Yaskawa INFORM job: A_ROOF_UPPER_0614_2_PAINT_52.JBI

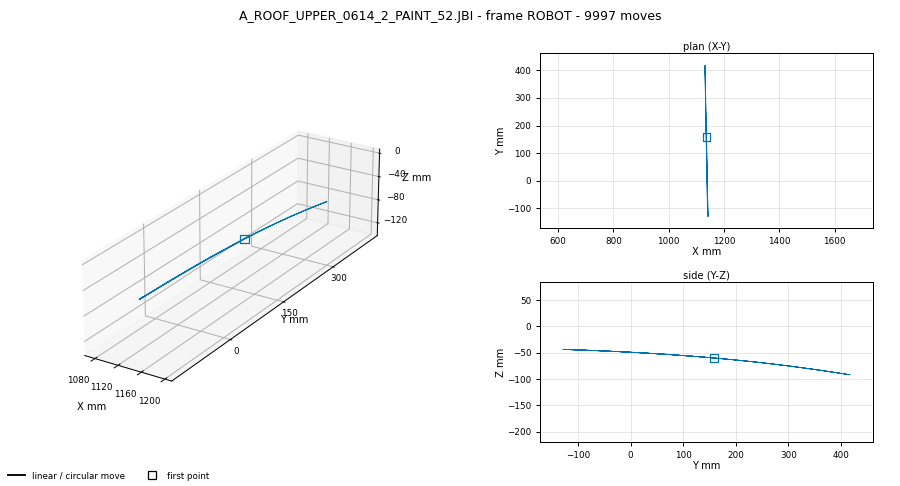
[picture p0: tool path of A_ROOF_UPPER_0614_2_PAINT_52.JBI in frame ROBOT, 9997 of 9997 moves have a stored position in this frame; points joined in program order, loops and branches not executed]
/JOB
//NAME A_ROOF_UPPER_0614_2_PAINT52
//POS
///NPOS 9997,0,0,0,0,0
///TOOL 1
///USER 0
///POSTYPE ROBOT
///RECTAN
///RCONF 1,0,0,0,0,0,0,0,0,0,0,0,0,0,0,0,0,0,0,0,0,0,0,0
C00000=1136.806,158.945,-59.840,-178.647,7.166,148.946
C00001=1136.811,158.695,-59.818,-178.650,7.165,148.946
C00002=1136.815,158.447,-59.796,-178.653,7.163,148.946
C00003=1136.820,158.198,-59.775,-178.656,7.160,148.947
C00004=1136.825,157.948,-59.753,-178.658,7.158,148.947
C00005=1136.829,157.680,-59.730,-178.662,7.156,148.947
C00006=1136.835,157.410,-59.707,-178.665,7.153,148.948
C00007=1136.840,157.141,-59.683,-178.668,7.152,148.948
C00008=1136.845,156.872,-59.660,-178.671,7.149,148.948
C00009=1136.850,156.623,-59.639,-178.674,7.147,148.949
C00010=1136.855,156.374,-59.617,-178.677,7.144,148.949
C00011=1136.859,156.125,-59.595,-178.679,7.143,148.949
C00012=1136.864,155.876,-59.573,-178.682,7.141,148.950
C00013=1136.869,155.627,-59.552,-178.685,7.139,148.950
C00014=1136.873,155.379,-59.531,-178.688,7.136,148.950
C00015=1136.878,155.129,-59.510,-178.690,7.135,148.951
C00016=1136.883,154.880,-59.488,-178.694,7.132,148.951
C00017=1136.887,154.632,-59.467,-178.696,7.131,148.951
C00018=1136.892,154.382,-59.445,-178.699,7.129,148.952
C00019=1136.897,154.133,-59.424,-178.702,7.126,148.952
C00020=1136.901,153.884,-59.403,-178.705,7.124,148.952
C00021=1136.906,153.635,-59.381,-178.707,7.123,148.953
C00022=1136.911,153.386,-59.359,-178.711,7.120,148.953
C00023=1136.916,153.137,-59.338,-178.713,7.118,148.953
C00024=1136.921,152.888,-59.317,-178.716,7.115,148.954
C00025=1136.925,152.639,-59.296,-178.719,7.114,148.954
C00026=1136.929,152.390,-59.274,-178.722,7.112,148.954
C00027=1136.934,152.141,-59.253,-178.725,7.110,148.955
C00028=1136.939,151.892,-59.232,-178.728,7.108,148.955
C00029=1136.944,151.643,-59.211,-178.730,7.106,148.955
C00030=1136.948,151.393,-59.190,-178.732,7.104,148.956
C00031=1136.953,151.144,-59.168,-178.736,7.102,148.956
C00032=1136.958,150.895,-59.147,-178.739,7.100,148.956
C00033=1136.962,150.647,-59.126,-178.741,7.098,148.957
C00034=1136.968,150.398,-59.105,-178.744,7.095,148.957
C00035=1136.972,150.148,-59.083,-178.747,7.094,148.957
C00036=1136.977,149.899,-59.062,-178.749,7.092,148.958
C00037=1136.982,149.650,-59.042,-178.753,7.089,148.958
C00038=1136.986,149.401,-59.020,-178.755,7.088,148.958
C00039=1136.992,149.152,-58.999,-178.758,7.086,148.959
C00040=1136.996,148.903,-58.979,-178.761,7.083,148.959
C00041=1137.000,148.654,-58.957,-178.764,7.081,148.959
C00042=1137.005,148.405,-58.936,-178.766,7.080,148.960
C00043=1137.010,148.156,-58.915,-178.770,7.077,148.960
C00044=1137.015,147.907,-58.894,-178.772,7.075,148.960
C00045=1137.020,147.658,-58.873,-178.775,7.073,148.961
C00046=1137.024,147.409,-58.852,-178.777,7.072,148.961
C00047=1137.029,147.159,-58.831,-178.781,7.069,148.961
C00048=1137.033,146.911,-58.810,-178.783,7.067,148.962
C00049=1137.038,146.661,-58.789,-178.786,7.066,148.962
C00050=1137.043,146.412,-58.768,-178.790,7.063,148.963
C00051=1137.048,146.163,-58.748,-178.792,7.062,148.963
C00052=1137.053,145.914,-58.727,-178.794,7.059,148.963
C00053=1137.057,145.665,-58.706,-178.797,7.058,148.963
C00054=1137.062,145.416,-58.685,-178.800,7.055,148.964
C00055=1137.067,145.167,-58.664,-178.803,7.054,148.964
C00056=1137.071,144.917,-58.643,-178.806,7.052,148.965
C00057=1137.076,144.668,-58.623,-178.809,7.049,148.965
C00058=1137.081,144.419,-58.602,-178.812,7.048,148.965
C00059=1137.085,144.170,-58.581,-178.814,7.046,148.966
C00060=1137.090,143.922,-58.560,-178.817,7.044,148.966
C00061=1137.095,143.673,-58.539,-178.820,7.041,148.966
C00062=1137.100,143.423,-58.518,-178.823,7.040,148.967
C00063=1137.104,143.174,-58.498,-178.826,7.038,148.967
C00064=1137.110,142.925,-58.477,-178.828,7.036,148.967
C00065=1137.114,142.676,-58.457,-178.832,7.034,148.968
C00066=1137.119,142.427,-58.436,-178.834,7.032,148.968
C00067=1137.124,142.178,-58.415,-178.837,7.030,148.968
C00068=1137.129,141.929,-58.394,-178.839,7.028,148.969
C00069=1137.133,141.680,-58.374,-178.843,7.026,148.969
C00070=1137.138,141.431,-58.354,-178.845,7.024,148.970
C00071=1137.143,141.182,-58.333,-178.848,7.022,148.970
C00072=1137.147,140.933,-58.312,-178.851,7.021,148.970
C00073=1137.152,140.683,-58.291,-178.854,7.018,148.971
C00074=1137.157,140.434,-58.271,-178.857,7.016,148.971
C00075=1137.161,140.185,-58.250,-178.859,7.014,148.971
C00076=1137.166,139.936,-58.230,-178.862,7.013,148.972
C00077=1137.171,139.687,-58.210,-178.865,7.010,148.972
C00078=1137.176,139.438,-58.189,-178.868,7.009,148.972
C00079=1137.181,139.188,-58.169,-178.871,7.007,148.973
C00080=1137.185,138.939,-58.148,-178.873,7.005,148.973
C00081=1137.190,138.690,-58.128,-178.877,7.003,148.974
C00082=1137.195,138.441,-58.107,-178.879,7.001,148.974
C00083=1137.199,138.192,-58.086,-178.882,6.999,148.974
C00084=1137.204,137.943,-58.067,-178.885,6.998,148.975
C00085=1137.209,137.693,-58.046,-178.887,6.995,148.975
C00086=1137.214,137.444,-58.025,-178.890,6.993,148.975
C00087=1137.218,137.196,-58.005,-178.893,6.991,148.976
C00088=1137.223,136.946,-57.984,-178.896,6.990,148.976
C00089=1137.228,136.697,-57.964,-178.898,6.988,148.977
C00090=1137.232,136.448,-57.944,-178.901,6.986,148.977
C00091=1137.237,136.199,-57.924,-178.905,6.984,148.977
C00092=1137.243,135.950,-57.903,-178.907,6.982,148.978
C00093=1137.247,135.701,-57.883,-178.910,6.980,148.978
C00094=1137.252,135.452,-57.863,-178.913,6.979,148.978
C00095=1137.256,135.203,-57.843,-178.915,6.977,148.979
C00096=1137.261,134.953,-57.823,-178.919,6.974,148.979
C00097=1137.266,134.704,-57.802,-178.921,6.972,148.979
C00098=1137.271,134.455,-57.782,-178.924,6.971,148.980
C00099=1137.275,134.205,-57.762,-178.926,6.969,148.980
C00100=1137.280,133.957,-57.742,-178.929,6.967,148.981
C00101=1137.285,133.708,-57.722,-178.932,6.965,148.981
C00102=1137.290,133.458,-57.701,-178.935,6.963,148.981
C00103=1137.295,133.209,-57.681,-178.938,6.961,148.982
C00104=1137.300,132.960,-57.661,-178.941,6.960,148.982
C00105=1137.304,132.711,-57.641,-178.943,6.958,148.983
C00106=1137.309,132.461,-57.621,-178.947,6.955,148.983
C00107=1137.314,132.213,-57.601,-178.949,6.954,148.983
C00108=1137.319,131.964,-57.580,-178.952,6.952,148.984
C00109=1137.324,131.695,-57.559,-178.955,6.950,148.984
C00110=1137.329,131.427,-57.538,-178.958,6.948,148.985
C00111=1137.334,131.158,-57.516,-178.961,6.946,148.985
C00112=1137.339,130.890,-57.495,-178.964,6.944,148.985
C00113=1137.344,130.640,-57.475,-178.967,6.942,148.986
C00114=1137.348,130.391,-57.455,-178.970,6.940,148.986
C00115=1137.354,130.142,-57.435,-178.972,6.939,148.986
C00116=1137.359,129.893,-57.414,-178.975,6.937,148.987
C00117=1137.363,129.643,-57.395,-178.978,6.935,148.987
C00118=1137.368,129.394,-57.374,-178.980,6.933,148.988
C00119=1137.373,129.145,-57.355,-178.984,6.931,148.988
C00120=1137.378,128.896,-57.335,-178.987,6.929,148.988
C00121=1137.382,128.647,-57.315,-178.989,6.928,148.989
C00122=1137.387,128.397,-57.295,-178.992,6.926,148.989
C00123=1137.392,128.148,-57.276,-178.995,6.924,148.990
C00124=1137.397,127.900,-57.256,-178.997,6.923,148.990
C00125=1137.402,127.650,-57.236,-179.000,6.921,148.990
C00126=1137.406,127.401,-57.216,-179.003,6.918,148.991
C00127=1137.411,127.152,-57.196,-179.006,6.917,148.991
C00128=1137.416,126.903,-57.177,-179.009,6.915,148.992
C00129=1137.421,126.653,-57.157,-179.012,6.913,148.992
C00130=1137.425,126.404,-57.137,-179.014,6.912,148.992
C00131=1137.431,126.155,-57.117,-179.017,6.910,148.993
C00132=1137.435,125.906,-57.098,-179.020,6.908,148.993
C00133=1137.439,125.657,-57.078,-179.023,6.907,148.994
C00134=1137.444,125.408,-57.059,-179.026,6.904,148.994
C00135=1137.449,125.159,-57.039,-179.029,6.902,148.994
C00136=1137.454,124.909,-57.019,-179.031,6.901,148.995
C00137=1137.459,124.659,-57.000,-179.034,6.899,148.995
C00138=1137.464,124.411,-56.980,-179.037,6.897,148.996
C00139=1137.468,124.162,-56.960,-179.039,6.896,148.996
C00140=1137.473,123.912,-56.940,-179.042,6.894,148.996
C00141=1137.478,123.664,-56.922,-179.045,6.892,148.997
C00142=1137.483,123.414,-56.902,-179.048,6.890,148.997
C00143=1137.488,123.165,-56.883,-179.051,6.888,148.998
C00144=1137.492,122.916,-56.862,-179.054,6.886,148.998
C00145=1137.497,122.667,-56.843,-179.056,6.885,148.998
C00146=1137.502,122.418,-56.824,-179.059,6.883,148.999
C00147=1137.506,122.168,-56.804,-179.062,6.881,148.999
C00148=1137.511,121.919,-56.785,-179.065,6.880,149.000
C00149=1137.517,121.670,-56.766,-179.067,6.878,149.000
C00150=1137.521,121.420,-56.746,-179.070,6.876,149.000
C00151=1137.526,121.171,-56.726,-179.073,6.875,149.001
C00152=1137.531,120.922,-56.708,-179.076,6.873,149.001
C00153=1137.535,120.673,-56.688,-179.079,6.870,149.002
C00154=1137.541,120.424,-56.669,-179.082,6.869,149.002
C00155=1137.545,120.174,-56.649,-179.084,6.867,149.002
C00156=1137.550,119.926,-56.630,-179.087,6.865,149.003
C00157=1137.555,119.676,-56.611,-179.090,6.864,149.003
C00158=1137.560,119.427,-56.591,-179.092,6.862,149.004
C00159=1137.565,119.178,-56.572,-179.095,6.860,149.004
C00160=1137.569,118.929,-56.553,-179.098,6.859,149.004
C00161=1137.574,118.680,-56.533,-179.101,6.857,149.005
C00162=1137.579,118.430,-56.514,-179.103,6.855,149.005
C00163=1137.584,118.182,-56.495,-179.106,6.853,149.006
C00164=1137.588,117.932,-56.475,-179.109,6.852,149.006
C00165=1137.594,117.683,-56.456,-179.112,6.850,149.006
C00166=1137.598,117.433,-56.438,-179.114,6.848,149.007
C00167=1137.603,117.184,-56.418,-179.117,6.847,149.007
C00168=1137.608,116.935,-56.399,-179.120,6.844,149.008
C00169=1137.612,116.686,-56.380,-179.123,6.843,149.008
C00170=1137.617,116.437,-56.360,-179.126,6.841,149.008
C00171=1137.622,116.187,-56.341,-179.129,6.839,149.009
C00172=1137.627,115.938,-56.323,-179.131,6.838,149.009
C00173=1137.632,115.688,-56.303,-179.134,6.836,149.010
C00174=1137.637,115.439,-56.284,-179.137,6.834,149.010
C00175=1137.641,115.190,-56.265,-179.139,6.832,149.011
C00176=1137.647,114.941,-56.245,-179.143,6.831,149.011
C00177=1137.651,114.691,-56.227,-179.145,6.829,149.012
C00178=1137.656,114.443,-56.208,-179.148,6.828,149.012
C00179=1137.662,114.194,-56.188,-179.151,6.826,149.012
C00180=1137.666,113.944,-56.170,-179.154,6.824,149.013
C00181=1137.671,113.695,-56.151,-179.156,6.823,149.013
C00182=1137.675,113.446,-56.132,-179.159,6.821,149.014
C00183=1137.681,113.197,-56.112,-179.162,6.819,149.014
C00184=1137.685,112.947,-56.094,-179.165,6.818,149.014
C00185=1137.690,112.698,-56.075,-179.167,6.816,149.015
C00186=1137.694,112.449,-56.056,-179.170,6.814,149.015
C00187=1137.700,112.199,-56.037,-179.173,6.813,149.016
C00188=1137.704,111.951,-56.018,-179.175,6.811,149.016
C00189=1137.710,111.701,-56.000,-179.178,6.809,149.016
C00190=1137.714,111.452,-55.981,-179.181,6.808,149.017
C00191=1137.719,111.203,-55.961,-179.184,6.806,149.017
C00192=1137.724,110.953,-55.943,-179.187,6.805,149.018
C00193=1137.729,110.704,-55.924,-179.190,6.803,149.018
C00194=1137.733,110.455,-55.906,-179.192,6.801,149.019
C00195=1137.739,110.206,-55.886,-179.195,6.800,149.019
C00196=1137.743,109.956,-55.868,-179.198,6.798,149.020
C00197=1137.748,109.707,-55.849,-179.200,6.796,149.020
C00198=1137.753,109.458,-55.830,-179.203,6.795,149.020
C00199=1137.758,109.208,-55.811,-179.206,6.793,149.021
C00200=1137.763,108.960,-55.792,-179.209,6.791,149.021
C00201=1137.768,108.711,-55.774,-179.211,6.789,149.022
C00202=1137.772,108.461,-55.755,-179.214,6.788,149.022
C00203=1137.777,108.212,-55.737,-179.217,6.786,149.022
C00204=1137.782,107.962,-55.718,-179.220,6.785,149.023
C00205=1137.787,107.713,-55.699,-179.223,6.783,149.023
C00206=1137.792,107.464,-55.681,-179.226,6.781,149.024
C00207=1137.797,107.214,-55.661,-179.228,6.780,149.024
C00208=1137.801,106.965,-55.643,-179.231,6.778,149.025
C00209=1137.806,106.717,-55.625,-179.234,6.776,149.025
C00210=1137.812,106.467,-55.606,-179.236,6.775,149.026
C00211=1137.816,106.217,-55.588,-179.239,6.773,149.026
C00212=1137.821,105.969,-55.569,-179.242,6.771,149.026
C00213=1137.826,105.700,-55.549,-179.245,6.770,149.027
C00214=1137.831,105.431,-55.529,-179.248,6.768,149.027
C00215=1137.837,105.163,-55.509,-179.251,6.766,149.028
C00216=1137.842,104.895,-55.489,-179.254,6.764,149.028
C00217=1137.846,104.646,-55.471,-179.257,6.763,149.029
C00218=1137.852,104.396,-55.453,-179.260,6.761,149.029
C00219=1137.856,104.147,-55.434,-179.263,6.760,149.030
C00220=1137.861,103.898,-55.416,-179.265,6.758,149.030
C00221=1137.867,103.648,-55.397,-179.268,6.757,149.030
C00222=1137.871,103.398,-55.379,-179.270,6.755,149.031
C00223=1137.876,103.150,-55.360,-179.273,6.754,149.031
C00224=1137.880,102.901,-55.342,-179.276,6.752,149.032
C00225=1137.885,102.652,-55.324,-179.278,6.750,149.032
C00226=1137.891,102.402,-55.305,-179.282,6.749,149.033
C00227=1137.895,102.152,-55.287,-179.284,6.747,149.033
C00228=1137.900,101.904,-55.268,-179.287,6.746,149.034
C00229=1137.905,101.654,-55.250,-179.290,6.744,149.034
C00230=1137.910,101.405,-55.232,-179.293,6.742,149.034
C00231=1137.915,101.155,-55.214,-179.295,6.741,149.035
C00232=1137.920,100.906,-55.196,-179.298,6.739,149.035
C00233=1137.925,100.657,-55.178,-179.301,6.737,149.036
C00234=1137.929,100.408,-55.159,-179.304,6.736,149.036
C00235=1137.934,100.159,-55.141,-179.307,6.734,149.037
C00236=1137.939,99.909,-55.123,-179.309,6.733,149.037
C00237=1137.944,99.660,-55.104,-179.312,6.732,149.038
C00238=1137.949,99.410,-55.086,-179.314,6.730,149.038
C00239=1137.954,99.161,-55.068,-179.317,6.728,149.038
C00240=1137.959,98.912,-55.050,-179.320,6.727,149.039
C00241=1137.964,98.663,-55.032,-179.323,6.725,149.039
C00242=1137.968,98.413,-55.014,-179.326,6.724,149.040
C00243=1137.973,98.164,-54.996,-179.329,6.722,149.040
C00244=1137.978,97.915,-54.978,-179.331,6.720,149.041
C00245=1137.983,97.666,-54.960,-179.334,6.719,149.041
C00246=1137.988,97.416,-54.942,-179.337,6.717,149.042
C00247=1137.993,97.167,-54.923,-179.339,6.716,149.042
C00248=1137.998,96.918,-54.905,-179.342,6.715,149.043
C00249=1138.003,96.668,-54.887,-179.345,6.713,149.043
C00250=1138.008,96.419,-54.869,-179.348,6.712,149.043
C00251=1138.012,96.169,-54.851,-179.350,6.710,149.044
C00252=1138.017,95.920,-54.833,-179.353,6.708,149.044
C00253=1138.022,95.671,-54.815,-179.356,6.707,149.045
C00254=1138.027,95.422,-54.797,-179.359,6.705,149.045
C00255=1138.032,95.173,-54.779,-179.362,6.704,149.046
C00256=1138.037,94.924,-54.761,-179.364,6.703,149.046
C00257=1138.042,94.674,-54.744,-179.367,6.701,149.047
C00258=1138.047,94.425,-54.726,-179.369,6.699,149.047
C00259=1138.051,94.175,-54.707,-179.372,6.698,149.047
C00260=1138.056,93.926,-54.689,-179.375,6.696,149.048
C00261=1138.061,93.676,-54.672,-179.378,6.695,149.048
C00262=1138.066,93.427,-54.654,-179.381,6.693,149.049
C00263=1138.071,93.177,-54.636,-179.384,6.691,149.049
C00264=1138.076,92.929,-54.619,-179.386,6.691,149.050
C00265=1138.080,92.679,-54.601,-179.388,6.689,149.050
C00266=1138.085,92.430,-54.583,-179.391,6.687,149.051
C00267=1138.090,92.181,-54.565,-179.394,6.686,149.051
C00268=1138.096,91.931,-54.548,-179.397,6.684,149.052
C00269=1138.100,91.682,-54.530,-179.400,6.683,149.052
C00270=1138.105,91.433,-54.512,-179.403,6.681,149.053
C00271=1138.110,91.184,-54.494,-179.405,6.680,149.053
C00272=1138.115,90.934,-54.476,-179.408,6.678,149.053
C00273=1138.120,90.685,-54.458,-179.411,6.677,149.054
C00274=1138.125,90.436,-54.441,-179.413,6.675,149.054
C00275=1138.130,90.186,-54.424,-179.416,6.674,149.055
C00276=1138.135,89.937,-54.406,-179.419,6.672,149.055
C00277=1138.140,89.688,-54.388,-179.422,6.670,149.056
C00278=1138.145,89.438,-54.371,-179.424,6.670,149.056
C00279=1138.150,89.189,-54.353,-179.427,6.668,149.057
C00280=1138.154,88.940,-54.335,-179.430,6.667,149.057
C00281=1138.159,88.690,-54.318,-179.433,6.665,149.058
C00282=1138.164,88.441,-54.300,-179.435,6.663,149.058
C00283=1138.169,88.191,-54.283,-179.438,6.662,149.058
C00284=1138.174,87.942,-54.265,-179.441,6.661,149.059
C00285=1138.178,87.693,-54.247,-179.443,6.659,149.060
C00286=1138.184,87.443,-54.230,-179.446,6.658,149.060
C00287=1138.188,87.194,-54.212,-179.449,6.656,149.060
C00288=1138.194,86.944,-54.195,-179.452,6.654,149.061
C00289=1138.199,86.695,-54.177,-179.455,6.653,149.061
C00290=1138.203,86.446,-54.160,-179.457,6.652,149.062
C00291=1138.208,86.196,-54.142,-179.460,6.651,149.062
C00292=1138.214,85.947,-54.125,-179.462,6.649,149.063
C00293=1138.218,85.699,-54.108,-179.465,6.647,149.063
C00294=1138.223,85.449,-54.091,-179.468,6.646,149.064
C00295=1138.228,85.200,-54.073,-179.471,6.645,149.064
C00296=1138.233,84.950,-54.055,-179.473,6.644,149.065
C00297=1138.238,84.701,-54.038,-179.476,6.642,149.065
C00298=1138.243,84.451,-54.021,-179.479,6.640,149.065
C00299=1138.248,84.202,-54.003,-179.482,6.639,149.066
C00300=1138.252,83.952,-53.986,-179.484,6.638,149.067
C00301=1138.257,83.703,-53.969,-179.487,6.636,149.067
C00302=1138.263,83.454,-53.951,-179.490,6.635,149.067
C00303=1138.267,83.205,-53.935,-179.492,6.633,149.068
C00304=1138.272,82.956,-53.917,-179.496,6.632,149.068
C00305=1138.277,82.706,-53.899,-179.498,6.631,149.069
C00306=1138.282,82.456,-53.883,-179.501,6.629,149.069
C00307=1138.287,82.207,-53.865,-179.503,6.628,149.070
C00308=1138.291,81.958,-53.848,-179.506,6.626,149.070
C00309=1138.297,81.708,-53.831,-179.509,6.625,149.071
C00310=1138.302,81.459,-53.813,-179.511,6.624,149.071
C00311=1138.307,81.210,-53.796,-179.514,6.622,149.072
C00312=1138.312,80.960,-53.779,-179.517,6.620,149.072
C00313=1138.316,80.711,-53.762,-179.520,6.619,149.073
C00314=1138.322,80.462,-53.745,-179.522,6.618,149.073
C00315=1138.327,80.212,-53.728,-179.525,6.617,149.074
C00316=1138.331,79.963,-53.711,-179.528,6.615,149.074
C00317=1138.337,79.694,-53.692,-179.531,6.614,149.075
C00318=1138.342,79.427,-53.674,-179.534,6.612,149.075
C00319=1138.347,79.158,-53.655,-179.537,6.611,149.076
C00320=1138.353,78.889,-53.636,-179.540,6.609,149.076
C00321=1138.358,78.640,-53.620,-179.542,6.607,149.077
C00322=1138.363,78.390,-53.603,-179.545,6.607,149.077
C00323=1138.367,78.141,-53.586,-179.548,6.605,149.078
C00324=1138.373,77.891,-53.569,-179.551,6.604,149.078
C00325=1138.377,77.643,-53.552,-179.553,6.602,149.079
C00326=1138.383,77.393,-53.535,-179.555,6.601,149.079
C00327=1138.387,77.144,-53.518,-179.559,6.600,149.080
C00328=1138.392,76.894,-53.501,-179.561,6.598,149.080
C00329=1138.397,76.645,-53.484,-179.564,6.597,149.081
C00330=1138.403,76.395,-53.467,-179.566,6.596,149.081
C00331=1138.407,76.146,-53.451,-179.569,6.594,149.081
C00332=1138.412,75.896,-53.434,-179.572,6.593,149.082
C00333=1138.417,75.648,-53.416,-179.575,6.591,149.082
C00334=1138.422,75.398,-53.400,-179.577,6.590,149.083
C00335=1138.427,75.149,-53.382,-179.580,6.589,149.083
C00336=1138.432,74.900,-53.366,-179.583,6.587,149.084
C00337=1138.436,74.650,-53.349,-179.585,6.586,149.084
C00338=1138.442,74.400,-53.332,-179.588,6.585,149.085
C00339=1138.446,74.151,-53.315,-179.591,6.583,149.085
C00340=1138.452,73.902,-53.299,-179.594,6.582,149.086
C00341=1138.456,73.652,-53.282,-179.596,6.581,149.086
C00342=1138.461,73.403,-53.265,-179.599,6.579,149.087
C00343=1138.467,73.154,-53.248,-179.602,6.578,149.087
C00344=1138.471,72.904,-53.232,-179.605,6.576,149.088
C00345=1138.476,72.655,-53.215,-179.607,6.576,149.088
C00346=1138.481,72.406,-53.198,-179.610,6.574,149.089
C00347=1138.486,72.156,-53.182,-179.613,6.572,149.089
C00348=1138.491,71.906,-53.165,-179.615,6.572,149.090
C00349=1138.496,71.657,-53.149,-179.618,6.570,149.090
C00350=1138.501,71.408,-53.132,-179.621,6.568,149.091
C00351=1138.505,71.158,-53.115,-179.623,6.568,149.091
C00352=1138.511,70.909,-53.098,-179.626,6.566,149.092
C00353=1138.516,70.660,-53.082,-179.629,6.565,149.092
C00354=1138.521,70.411,-53.065,-179.632,6.563,149.093
C00355=1138.526,70.161,-53.048,-179.634,6.562,149.093
C00356=1138.531,69.911,-53.032,-179.637,6.561,149.094
C00357=1138.536,69.662,-53.016,-179.640,6.559,149.094
C00358=1138.540,69.413,-52.999,-179.642,6.558,149.095
C00359=1138.546,69.164,-52.982,-179.645,6.557,149.095
C00360=1138.551,68.914,-52.966,-179.648,6.555,149.096
C00361=1138.555,68.664,-52.950,-179.650,6.555,149.096
C00362=1138.561,68.415,-52.933,-179.653,6.553,149.097
C00363=1138.566,68.165,-52.916,-179.656,6.552,149.097
C00364=1138.571,67.917,-52.900,-179.658,6.551,149.098
C00365=1138.575,67.667,-52.883,-179.661,6.549,149.098
C00366=1138.580,67.417,-52.867,-179.664,6.547,149.099
C00367=1138.585,67.168,-52.851,-179.666,6.547,149.099
C00368=1138.590,66.918,-52.834,-179.669,6.545,149.100
C00369=1138.596,66.669,-52.818,-179.672,6.544,149.100
C00370=1138.600,66.420,-52.801,-179.674,6.543,149.101
C00371=1138.605,66.171,-52.785,-179.677,6.542,149.101
C00372=1138.610,65.921,-52.768,-179.680,6.540,149.102
C00373=1138.615,65.671,-52.752,-179.682,6.539,149.102
C00374=1138.620,65.422,-52.735,-179.685,6.538,149.103
C00375=1138.625,65.172,-52.719,-179.688,6.536,149.103
C00376=1138.630,64.923,-52.703,-179.690,6.535,149.104
C00377=1138.635,64.674,-52.687,-179.693,6.534,149.104
C00378=1138.640,64.424,-52.671,-179.696,6.532,149.105
C00379=1138.645,64.175,-52.654,-179.698,6.532,149.105
C00380=1138.650,63.926,-52.638,-179.701,6.530,149.106
C00381=1138.655,63.676,-52.622,-179.704,6.529,149.106
C00382=1138.660,63.427,-52.606,-179.706,6.528,149.107
C00383=1138.665,63.177,-52.589,-179.709,6.526,149.107
C00384=1138.670,62.928,-52.573,-179.712,6.524,149.108
C00385=1138.675,62.678,-52.557,-179.715,6.524,149.108
C00386=1138.680,62.429,-52.541,-179.717,6.522,149.109
C00387=1138.685,62.180,-52.524,-179.720,6.521,149.109
C00388=1138.690,61.930,-52.508,-179.723,6.520,149.110
C00389=1138.694,61.681,-52.492,-179.725,6.519,149.110
C00390=1138.700,61.431,-52.476,-179.728,6.518,149.111
C00391=1138.704,61.182,-52.459,-179.730,6.516,149.111
C00392=1138.710,60.932,-52.444,-179.734,6.515,149.112
C00393=1138.715,60.683,-52.428,-179.736,6.514,149.112
C00394=1138.720,60.433,-52.412,-179.739,6.512,149.113
C00395=1138.725,60.184,-52.396,-179.742,6.511,149.113
C00396=1138.729,59.935,-52.379,-179.744,6.510,149.114
C00397=1138.735,59.685,-52.364,-179.747,6.509,149.114
C00398=1138.739,59.436,-52.347,-179.749,6.508,149.115
C00399=1138.745,59.186,-52.331,-179.752,6.506,149.115
C00400=1138.750,58.937,-52.316,-179.755,6.505,149.116
C00401=1138.755,58.687,-52.299,-179.757,6.504,149.116
C00402=1138.760,58.438,-52.284,-179.760,6.503,149.117
C00403=1138.764,58.189,-52.267,-179.763,6.501,149.117
C00404=1138.770,57.939,-52.251,-179.765,6.500,149.118
C00405=1138.775,57.690,-52.236,-179.768,6.499,149.118
C00406=1138.780,57.440,-52.219,-179.770,6.498,149.119
C00407=1138.785,57.191,-52.204,-179.773,6.496,149.119
C00408=1138.789,56.941,-52.188,-179.776,6.495,149.120
C00409=1138.794,56.692,-52.172,-179.779,6.494,149.120
C00410=1138.800,56.443,-52.156,-179.781,6.493,149.121
C00411=1138.804,56.193,-52.140,-179.784,6.492,149.121
C00412=1138.810,55.943,-52.125,-179.787,6.491,149.122
C00413=1138.815,55.695,-52.108,-179.789,6.490,149.122
C00414=1138.820,55.444,-52.092,-179.792,6.488,149.123
C00415=1138.825,55.195,-52.077,-179.795,6.487,149.123
C00416=1138.830,54.946,-52.061,-179.797,6.486,149.124
C00417=1138.834,54.696,-52.045,-179.800,6.484,149.124
C00418=1138.839,54.447,-52.030,-179.802,6.484,149.125
C00419=1138.845,54.198,-52.014,-179.805,6.482,149.125
C00420=1138.850,53.948,-51.998,-179.808,6.481,149.126
C00421=1138.855,53.679,-51.981,-179.811,6.480,149.127
C00422=1138.861,53.411,-51.964,-179.813,6.479,149.127
C00423=1138.866,53.142,-51.947,-179.817,6.477,149.128
C00424=1138.871,52.874,-51.931,-179.819,6.476,149.128
C00425=1138.876,52.624,-51.915,-179.822,6.475,149.129
C00426=1138.881,52.374,-51.899,-179.825,6.474,149.129
C00427=1138.887,52.125,-51.883,-179.827,6.473,149.130
C00428=1138.891,51.875,-51.868,-179.830,6.471,149.130
C00429=1138.896,51.626,-51.852,-179.832,6.471,149.131
C00430=1138.901,51.377,-51.836,-179.835,6.469,149.131
C00431=1138.907,51.128,-51.821,-179.838,6.467,149.132
C00432=1138.911,50.878,-51.805,-179.840,6.467,149.132
C00433=1138.916,50.628,-51.790,-179.843,6.465,149.133
C00434=1138.921,50.379,-51.774,-179.845,6.464,149.133
C00435=1138.927,50.130,-51.759,-179.849,6.463,149.134
C00436=1138.932,49.880,-51.743,-179.851,6.462,149.134
C00437=1138.936,49.630,-51.728,-179.854,6.461,149.135
C00438=1138.942,49.381,-51.712,-179.856,6.460,149.135
C00439=1138.947,49.132,-51.696,-179.859,6.459,149.136
C00440=1138.951,48.882,-51.681,-179.861,6.458,149.136
C00441=1138.956,48.632,-51.665,-179.864,6.456,149.137
C00442=1138.962,48.383,-51.650,-179.867,6.455,149.137
C00443=1138.966,48.134,-51.635,-179.869,6.454,149.138
C00444=1138.971,47.884,-51.619,-179.873,6.453,149.139
C00445=1138.977,47.634,-51.603,-179.875,6.452,149.139
C00446=1138.981,47.385,-51.588,-179.877,6.450,149.139
C00447=1138.987,47.136,-51.573,-179.880,6.449,149.140
C00448=1138.992,46.887,-51.557,-179.883,6.448,149.141
C00449=1138.996,46.637,-51.542,-179.885,6.447,149.141
C00450=1139.002,46.387,-51.526,-179.888,6.446,149.141
C00451=1139.006,46.138,-51.511,-179.890,6.445,149.142
C00452=1139.012,45.888,-51.496,-179.893,6.444,149.143
C00453=1139.017,45.639,-51.481,-179.895,6.443,149.143
C00454=1139.021,45.389,-51.465,-179.899,6.441,149.144
C00455=1139.027,45.140,-51.450,-179.901,6.441,149.144
C00456=1139.031,44.891,-51.435,-179.903,6.439,149.145
C00457=1139.037,44.641,-51.419,-179.906,6.439,149.145
C00458=1139.042,44.392,-51.404,-179.909,6.437,149.146
C00459=1139.047,44.142,-51.389,-179.911,6.436,149.146
C00460=1139.052,43.893,-51.374,-179.914,6.435,149.147
C00461=1139.056,43.643,-51.358,-179.916,6.434,149.147
C00462=1139.062,43.393,-51.343,-179.919,6.432,149.148
C00463=1139.067,43.144,-51.328,-179.922,6.432,149.148
C00464=1139.072,42.894,-51.313,-179.925,6.430,149.149
C00465=1139.077,42.645,-51.298,-179.927,6.429,149.149
C00466=1139.082,42.396,-51.282,-179.930,6.428,149.150
C00467=1139.087,42.147,-51.267,-179.932,6.427,149.150
C00468=1139.093,41.897,-51.253,-179.935,6.426,149.151
C00469=1139.097,41.647,-51.237,-179.938,6.425,149.151
C00470=1139.102,41.398,-51.222,-179.940,6.424,149.152
C00471=1139.107,41.148,-51.207,-179.943,6.423,149.153
C00472=1139.112,40.898,-51.192,-179.946,6.422,149.153
C00473=1139.117,40.649,-51.177,-179.948,6.421,149.153
C00474=1139.122,40.400,-51.161,-179.951,6.419,149.154
C00475=1139.127,40.150,-51.147,-179.953,6.419,149.155
C00476=1139.133,39.901,-51.131,-179.956,6.417,149.155
C00477=1139.138,39.651,-51.117,-179.959,6.417,149.156
C00478=1139.143,39.402,-51.101,-179.961,6.415,149.156
C00479=1139.148,39.153,-51.086,-179.964,6.414,149.157
C00480=1139.153,38.903,-51.072,-179.967,6.413,149.157
C00481=1139.158,38.654,-51.057,-179.969,6.412,149.158
C00482=1139.163,38.404,-51.042,-179.972,6.410,149.158
C00483=1139.168,38.154,-51.026,-179.974,6.410,149.159
C00484=1139.172,37.905,-51.011,-179.977,6.409,149.159
C00485=1139.178,37.655,-50.996,-179.979,6.407,149.160
C00486=1139.183,37.406,-50.981,-179.982,6.407,149.160
C00487=1139.188,37.156,-50.967,-179.985,6.405,149.161
C00488=1139.193,36.906,-50.952,-179.987,6.405,149.161
C00489=1139.198,36.657,-50.937,-179.990,6.403,149.162
C00490=1139.203,36.408,-50.922,-179.992,6.402,149.162
C00491=1139.208,36.158,-50.907,-179.995,6.401,149.163
C00492=1139.213,35.908,-50.892,-179.998,6.400,149.164
C00493=1139.218,35.659,-50.877,179.999,6.399,149.164
C00494=1139.223,35.409,-50.863,179.997,6.398,149.165
C00495=1139.228,35.160,-50.848,179.995,6.397,149.165
C00496=1139.234,34.910,-50.833,179.992,6.396,149.166
C00497=1139.239,34.661,-50.818,179.989,6.395,149.166
C00498=1139.243,34.411,-50.803,179.986,6.394,149.167
C00499=1139.248,34.162,-50.789,179.984,6.393,149.167
C00500=1139.254,33.912,-50.774,179.981,6.392,149.168
C00501=1139.259,33.663,-50.760,179.979,6.391,149.168
C00502=1139.264,33.414,-50.745,179.977,6.390,149.169
C00503=1139.270,33.164,-50.730,179.973,6.389,149.169
C00504=1139.275,32.915,-50.716,179.971,6.388,149.170
C00505=1139.279,32.665,-50.701,179.969,6.386,149.170
C00506=1139.284,32.416,-50.686,179.966,6.386,149.171
C00507=1139.290,32.166,-50.671,179.963,6.384,149.172
C00508=1139.295,31.917,-50.656,179.961,6.383,149.172
C00509=1139.299,31.667,-50.642,179.958,6.383,149.173
C00510=1139.304,31.418,-50.627,179.956,6.381,149.173
C00511=1139.310,31.168,-50.612,179.953,6.381,149.174
C00512=1139.315,30.918,-50.598,179.950,6.379,149.174
C00513=1139.319,30.669,-50.583,179.948,6.378,149.175
C00514=1139.324,30.419,-50.569,179.945,6.377,149.175
C00515=1139.329,30.170,-50.554,179.943,6.376,149.176
C00516=1139.336,29.920,-50.540,179.940,6.376,149.176
C00517=1139.340,29.671,-50.525,179.937,6.374,149.177
C00518=1139.345,29.421,-50.511,179.935,6.373,149.177
C00519=1139.350,29.172,-50.496,179.932,6.372,149.178
C00520=1139.355,28.922,-50.482,179.930,6.371,149.179
C00521=1139.360,28.673,-50.467,179.927,6.371,149.179
C00522=1139.365,28.423,-50.452,179.924,6.369,149.180
C00523=1139.370,28.173,-50.438,179.922,6.368,149.180
C00524=1139.376,27.924,-50.424,179.919,6.367,149.181
C00525=1139.381,27.655,-50.408,179.917,6.366,149.181
C00526=1139.386,27.387,-50.393,179.914,6.365,149.182
C00527=1139.392,27.117,-50.377,179.911,6.364,149.182
C00528=1139.398,26.848,-50.361,179.908,6.363,149.183
C00529=1139.403,26.598,-50.347,179.906,6.362,149.184
C00530=1139.407,26.349,-50.333,179.903,6.361,149.184
C00531=1139.413,26.100,-50.319,179.900,6.360,149.185
C00532=1139.418,25.851,-50.304,179.898,6.359,149.185
C00533=1139.423,25.601,-50.290,179.895,6.358,149.186
C00534=1139.428,25.351,-50.275,179.893,6.357,149.186
C00535=1139.433,25.101,-50.261,179.891,6.357,149.187
C00536=1139.437,24.852,-50.247,179.888,6.355,149.187
C00537=1139.444,24.602,-50.232,179.885,6.354,149.188
C00538=1139.449,24.353,-50.218,179.882,6.353,149.188
C00539=1139.454,24.103,-50.204,179.880,6.352,149.189
C00540=1139.459,23.853,-50.189,179.878,6.352,149.189
C00541=1139.464,23.604,-50.175,179.875,6.350,149.190
C00542=1139.469,23.355,-50.161,179.872,6.350,149.191
C00543=1139.474,23.105,-50.147,179.870,6.349,149.191
C00544=1139.479,22.855,-50.133,179.867,6.347,149.191
C00545=1139.484,22.605,-50.118,179.865,6.347,149.192
C00546=1139.490,22.356,-50.105,179.862,6.346,149.193
C00547=1139.495,22.107,-50.090,179.860,6.344,149.193
C00548=1139.499,21.857,-50.076,179.857,6.344,149.194
C00549=1139.504,21.607,-50.062,179.855,6.343,149.194
C00550=1139.509,21.358,-50.047,179.852,6.342,149.195
C00551=1139.515,21.109,-50.034,179.849,6.341,149.195
C00552=1139.519,20.859,-50.020,179.847,6.339,149.196
C00553=1139.524,20.609,-50.006,179.844,6.339,149.196
C00554=1139.530,20.360,-49.992,179.842,6.338,149.197
C00555=1139.535,20.111,-49.977,179.839,6.336,149.197
C00556=1139.540,19.861,-49.963,179.836,6.336,149.198
C00557=1139.545,19.611,-49.949,179.834,6.335,149.199
C00558=1139.550,19.362,-49.935,179.831,6.334,149.199
C00559=1139.555,19.113,-49.921,179.829,6.333,149.200
C00560=1139.560,18.862,-49.907,179.827,6.332,149.200
C00561=1139.566,18.613,-49.893,179.823,6.331,149.201
C00562=1139.571,18.364,-49.879,179.821,6.330,149.201
C00563=1139.576,18.114,-49.865,179.819,6.329,149.202
C00564=1139.581,17.864,-49.850,179.816,6.328,149.202
C00565=1139.586,17.615,-49.837,179.814,6.327,149.203
C00566=1139.591,17.366,-49.823,179.811,6.327,149.204
C00567=1139.596,17.115,-49.809,179.809,6.326,149.204
C00568=1139.601,16.866,-49.795,179.806,6.324,149.204
C00569=1139.606,16.617,-49.781,179.803,6.324,149.205
C00570=1139.611,16.367,-49.767,179.801,6.323,149.206
C00571=1139.616,16.118,-49.753,179.798,6.322,149.206
C00572=1139.621,15.868,-49.740,179.796,6.321,149.207
C00573=1139.626,15.618,-49.726,179.794,6.320,149.207
C00574=1139.632,15.369,-49.712,179.790,6.319,149.208
C00575=1139.637,15.119,-49.697,179.788,6.318,149.208
C00576=1139.642,14.869,-49.684,179.786,6.317,149.209
C00577=1139.647,14.620,-49.670,179.783,6.316,149.209
C00578=1139.652,14.371,-49.656,179.781,6.315,149.210
C00579=1139.658,14.121,-49.643,179.778,6.315,149.211
C00580=1139.663,13.871,-49.629,179.776,6.314,149.211
C00581=1139.667,13.622,-49.615,179.773,6.313,149.212
C00582=1139.673,13.372,-49.602,179.770,6.312,149.212
C00583=1139.678,13.123,-49.588,179.768,6.311,149.213
C00584=1139.683,12.873,-49.573,179.765,6.310,149.213
C00585=1139.688,12.623,-49.560,179.763,6.309,149.214
C00586=1139.693,12.374,-49.546,179.761,6.308,149.214
C00587=1139.698,12.125,-49.532,179.758,6.308,149.215
C00588=1139.704,11.875,-49.519,179.755,6.306,149.215
C00589=1139.708,11.625,-49.505,179.753,6.306,149.216
C00590=1139.713,11.376,-49.491,179.750,6.305,149.217
C00591=1139.719,11.126,-49.478,179.748,6.304,149.217
C00592=1139.724,10.877,-49.464,179.745,6.303,149.218
C00593=1139.729,10.627,-49.451,179.743,6.302,149.218
C00594=1139.734,10.378,-49.437,179.741,6.301,149.219
C00595=1139.739,10.128,-49.423,179.737,6.300,149.219
C00596=1139.744,9.879,-49.410,179.735,6.299,149.220
C00597=1139.749,9.629,-49.396,179.733,6.299,149.220
C00598=1139.754,9.379,-49.382,179.730,6.298,149.221
C00599=1139.759,9.130,-49.369,179.728,6.297,149.221
C00600=1139.765,8.880,-49.355,179.725,6.296,149.222
C00601=1139.770,8.631,-49.341,179.723,6.295,149.223
C00602=1139.775,8.381,-49.329,179.720,6.294,149.223
C00603=1139.780,8.132,-49.315,179.717,6.293,149.224
C00604=1139.785,7.881,-49.301,179.715,6.292,149.224
C00605=1139.790,7.633,-49.288,179.713,6.292,149.225
C00606=1139.796,7.382,-49.274,179.710,6.290,149.225
C00607=1139.800,7.134,-49.261,179.708,6.290,149.226
C00608=1139.806,6.883,-49.247,179.705,6.289,149.226
C00609=1139.811,6.634,-49.234,179.703,6.288,149.227
C00610=1139.816,6.384,-49.220,179.700,6.287,149.227
C00611=1139.822,6.135,-49.207,179.697,6.286,149.228
C00612=1139.826,5.885,-49.194,179.695,6.286,149.229
C00613=1139.832,5.636,-49.180,179.693,6.285,149.229
C00614=1139.837,5.386,-49.166,179.690,6.284,149.230
C00615=1139.842,5.137,-49.153,179.687,6.283,149.230
C00616=1139.847,4.886,-49.140,179.685,6.282,149.231
C00617=1139.852,4.638,-49.127,179.683,6.281,149.231
C00618=1139.857,4.387,-49.113,179.680,6.281,149.232
C00619=1139.862,4.138,-49.100,179.677,6.279,149.232
C00620=1139.867,3.888,-49.086,179.675,6.279,149.233
C00621=1139.872,3.639,-49.074,179.672,6.278,149.234
C00622=1139.878,3.389,-49.060,179.670,6.277,149.234
C00623=1139.882,3.140,-49.047,179.667,6.276,149.235
C00624=1139.888,2.890,-49.033,179.665,6.275,149.235
C00625=1139.893,2.640,-49.020,179.663,6.275,149.236
C00626=1139.898,2.391,-49.007,179.660,6.274,149.236
C00627=1139.903,2.141,-48.994,179.658,6.273,149.237
C00628=1139.909,1.892,-48.980,179.655,6.272,149.237
C00629=1139.913,1.622,-48.966,179.652,6.271,149.238
C00630=1139.919,1.352,-48.952,179.650,6.270,149.238
C00631=1139.925,1.083,-48.938,179.647,6.269,149.239
C00632=1139.930,0.814,-48.923,179.644,6.269,149.240
C00633=1139.936,0.564,-48.910,179.642,6.268,149.240
C00634=1139.941,0.314,-48.897,179.639,6.266,149.241
C00635=1139.946,0.065,-48.884,179.637,6.266,149.241
C00636=1139.951,-0.185,-48.870,179.634,6.265,149.242
C00637=1139.956,-0.434,-48.857,179.632,6.264,149.242
C00638=1139.962,-0.684,-48.845,179.630,6.264,149.243
C00639=1139.967,-0.934,-48.831,179.627,6.262,149.244
C00640=1139.972,-1.183,-48.818,179.624,6.262,149.244
C00641=1139.977,-1.432,-48.805,179.622,6.261,149.245
C00642=1139.982,-1.682,-48.792,179.620,6.260,149.245
C00643=1139.987,-1.932,-48.779,179.617,6.260,149.246
C00644=1139.992,-2.182,-48.766,179.614,6.258,149.246
C00645=1139.998,-2.431,-48.753,179.612,6.258,149.247
C00646=1140.003,-2.681,-48.740,179.610,6.257,149.247
C00647=1140.008,-2.931,-48.727,179.607,6.256,149.248
C00648=1140.013,-3.180,-48.714,179.605,6.256,149.249
C00649=1140.018,-3.430,-48.701,179.602,6.254,149.249
C00650=1140.023,-3.679,-48.687,179.600,6.253,149.250
C00651=1140.028,-3.929,-48.675,179.597,6.253,149.250
C00652=1140.033,-4.178,-48.662,179.595,6.252,149.251
C00653=1140.039,-4.428,-48.648,179.592,6.252,149.251
C00654=1140.044,-4.678,-48.636,179.590,6.251,149.252
C00655=1140.049,-4.927,-48.623,179.587,6.249,149.252
C00656=1140.054,-5.177,-48.610,179.585,6.249,149.253
C00657=1140.059,-5.427,-48.597,179.583,6.248,149.254
C00658=1140.064,-5.676,-48.584,179.580,6.248,149.254
C00659=1140.070,-5.925,-48.571,179.578,6.247,149.255
C00660=1140.075,-6.176,-48.558,179.575,6.246,149.255
C00661=1140.080,-6.425,-48.546,179.572,6.245,149.256
C00662=1140.085,-6.674,-48.533,179.570,6.244,149.256
C00663=1140.090,-6.924,-48.520,179.568,6.243,149.257
C00664=1140.095,-7.174,-48.507,179.565,6.243,149.257
C00665=1140.101,-7.423,-48.494,179.563,6.242,149.258
C00666=1140.106,-7.672,-48.482,179.560,6.242,149.259
C00667=1140.111,-7.923,-48.468,179.558,6.240,149.259
C00668=1140.116,-8.172,-48.456,179.555,6.239,149.260
C00669=1140.121,-8.421,-48.443,179.553,6.239,149.260
C00670=1140.127,-8.671,-48.431,179.551,6.238,149.261
C00671=1140.132,-8.922,-48.417,179.548,6.238,149.261
C00672=1140.137,-9.171,-48.405,179.546,6.237,149.262
C00673=1140.142,-9.420,-48.392,179.544,6.236,149.262
C00674=1140.147,-9.670,-48.380,179.540,6.235,149.263
C00675=1140.152,-9.920,-48.367,179.538,6.234,149.263
C00676=1140.158,-10.169,-48.354,179.536,6.233,149.264
C00677=1140.163,-10.419,-48.341,179.533,6.233,149.265
C00678=1140.168,-10.669,-48.329,179.531,6.232,149.265
C00679=1140.173,-10.919,-48.316,179.528,6.232,149.266
C00680=1140.178,-11.168,-48.303,179.526,6.231,149.266
C00681=1140.183,-11.417,-48.291,179.523,6.229,149.267
C00682=1140.188,-11.666,-48.278,179.521,6.229,149.267
C00683=1140.194,-11.916,-48.265,179.519,6.228,149.268
C00684=1140.199,-12.167,-48.253,179.516,6.228,149.269
C00685=1140.204,-12.416,-48.240,179.514,6.227,149.269
C00686=1140.209,-12.665,-48.228,179.512,6.226,149.270
C00687=1140.214,-12.915,-48.215,179.509,6.226,149.270
C00688=1140.220,-13.165,-48.203,179.507,6.225,149.271
C00689=1140.224,-13.415,-48.190,179.505,6.224,149.271
C00690=1140.229,-13.664,-48.178,179.501,6.223,149.272
C00691=1140.235,-13.914,-48.164,179.499,6.222,149.272
C00692=1140.240,-14.164,-48.152,179.497,6.222,149.273
C00693=1140.246,-14.413,-48.140,179.494,6.221,149.273
C00694=1140.251,-14.662,-48.127,179.492,6.220,149.274
C00695=1140.255,-14.912,-48.114,179.490,6.219,149.275
C00696=1140.261,-15.162,-48.102,179.487,6.219,149.275
C00697=1140.266,-15.411,-48.090,179.485,6.218,149.276
C00698=1140.271,-15.661,-48.077,179.482,6.217,149.276
C00699=1140.276,-15.911,-48.065,179.480,6.216,149.277
C00700=1140.281,-16.160,-48.053,179.477,6.215,149.277
C00701=1140.287,-16.409,-48.040,179.475,6.215,149.278
C00702=1140.291,-16.660,-48.028,179.473,6.214,149.278
C00703=1140.297,-16.909,-48.015,179.470,6.213,149.279
C00704=1140.302,-17.159,-48.003,179.468,6.213,149.280
C00705=1140.307,-17.409,-47.991,179.466,6.212,149.280
C00706=1140.312,-17.658,-47.978,179.463,6.211,149.281
C00707=1140.318,-17.908,-47.966,179.461,6.211,149.281
C00708=1140.323,-18.157,-47.954,179.458,6.210,149.282
C00709=1140.328,-18.407,-47.942,179.455,6.209,149.282
C00710=1140.333,-18.656,-47.929,179.453,6.208,149.283
C00711=1140.338,-18.906,-47.917,179.451,6.207,149.284
C00712=1140.343,-19.156,-47.904,179.448,6.207,149.284
C00713=1140.348,-19.406,-47.892,179.446,6.206,149.285
C00714=1140.354,-19.656,-47.880,179.443,6.205,149.285
C00715=1140.359,-19.905,-47.867,179.441,6.205,149.286
C00716=1140.364,-20.155,-47.855,179.439,6.204,149.286
C00717=1140.370,-20.404,-47.843,179.436,6.203,149.287
C00718=1140.375,-20.654,-47.831,179.434,6.203,149.287
C00719=1140.380,-20.903,-47.818,179.432,6.202,149.288
C00720=1140.386,-21.153,-47.806,179.429,6.201,149.288
C00721=1140.391,-21.403,-47.794,179.427,6.201,149.289
C00722=1140.396,-21.653,-47.782,179.425,6.200,149.290
C00723=1140.401,-21.902,-47.769,179.422,6.199,149.290
C00724=1140.407,-22.152,-47.757,179.419,6.198,149.291
C00725=1140.412,-22.401,-47.745,179.417,6.197,149.291
C00726=1140.417,-22.651,-47.733,179.415,6.197,149.292
C00727=1140.422,-22.900,-47.721,179.412,6.196,149.292
C00728=1140.427,-23.150,-47.709,179.410,6.195,149.293
C00729=1140.432,-23.400,-47.697,179.408,6.195,149.293
C00730=1140.438,-23.649,-47.685,179.405,6.194,149.294
C00731=1140.443,-23.899,-47.673,179.403,6.193,149.295
C00732=1140.448,-24.149,-47.660,179.400,6.193,149.295
C00733=1140.453,-24.419,-47.647,179.398,6.192,149.296
C00734=1140.459,-24.689,-47.634,179.395,6.192,149.296
C00735=1140.465,-24.959,-47.622,179.393,6.190,149.297
C00736=1140.471,-25.230,-47.608,179.390,6.190,149.298
C00737=1140.475,-25.479,-47.596,179.388,6.189,149.298
C00738=1140.480,-25.729,-47.584,179.385,6.189,149.299
C00739=1140.486,-25.978,-47.572,179.383,6.188,149.299
C00740=1140.491,-26.228,-47.560,179.381,6.187,149.300
C00741=1140.496,-26.478,-47.548,179.378,6.187,149.300
C00742=1140.501,-26.727,-47.536,179.376,6.186,149.301
C00743=1140.506,-26.977,-47.524,179.374,6.185,149.301
C00744=1140.512,-27.227,-47.512,179.371,6.185,149.302
C00745=1140.517,-27.477,-47.500,179.369,6.184,149.302
C00746=1140.523,-27.726,-47.488,179.366,6.184,149.303
C00747=1140.527,-27.975,-47.476,179.364,6.183,149.304
C00748=1140.532,-28.225,-47.464,179.362,6.182,149.304
C00749=1140.538,-28.475,-47.453,179.359,6.182,149.305
C00750=1140.544,-28.724,-47.440,179.357,6.181,149.305
C00751=1140.548,-28.974,-47.429,179.355,6.180,149.306
C00752=1140.554,-29.224,-47.417,179.352,6.180,149.306
C00753=1140.559,-29.473,-47.405,179.350,6.179,149.307
C00754=1140.565,-29.723,-47.393,179.348,6.178,149.307
C00755=1140.569,-29.972,-47.381,179.345,6.178,149.308
C00756=1140.574,-30.222,-47.369,179.343,6.177,149.309
C00757=1140.580,-30.472,-47.357,179.340,6.176,149.309
C00758=1140.584,-30.722,-47.346,179.338,6.176,149.310
C00759=1140.590,-30.972,-47.334,179.336,6.175,149.310
C00760=1140.595,-31.221,-47.322,179.333,6.174,149.311
C00761=1140.600,-31.471,-47.310,179.330,6.173,149.311
C00762=1140.606,-31.720,-47.299,179.328,6.172,149.312
C00763=1140.611,-31.970,-47.287,179.326,6.172,149.313
C00764=1140.617,-32.220,-47.275,179.323,6.171,149.313
C00765=1140.621,-32.470,-47.264,179.321,6.170,149.314
C00766=1140.627,-32.719,-47.252,179.319,6.170,149.314
C00767=1140.632,-32.969,-47.239,179.316,6.169,149.315
C00768=1140.637,-33.218,-47.228,179.314,6.168,149.315
C00769=1140.642,-33.468,-47.216,179.312,6.168,149.316
C00770=1140.648,-33.718,-47.205,179.310,6.168,149.316
C00771=1140.653,-33.967,-47.193,179.307,6.167,149.317
C00772=1140.658,-34.217,-47.181,179.305,6.166,149.318
C00773=1140.663,-34.467,-47.170,179.303,6.166,149.318
C00774=1140.668,-34.717,-47.158,179.300,6.165,149.319
C00775=1140.674,-34.967,-47.146,179.298,6.165,149.319
C00776=1140.679,-35.216,-47.136,179.296,6.164,149.320
C00777=1140.684,-35.465,-47.124,179.293,6.163,149.320
C00778=1140.690,-35.715,-47.112,179.291,6.163,149.321
C00779=1140.695,-35.965,-47.100,179.289,6.162,149.321
C00780=1140.700,-36.215,-47.089,179.286,6.161,149.322
C00781=1140.705,-36.465,-47.077,179.284,6.161,149.322
C00782=1140.711,-36.714,-47.066,179.281,6.160,149.323
C00783=1140.715,-36.963,-47.054,179.279,6.159,149.324
C00784=1140.721,-37.213,-47.043,179.277,6.159,149.324
C00785=1140.726,-37.463,-47.031,179.274,6.158,149.325
C00786=1140.731,-37.713,-47.019,179.272,6.157,149.325
C00787=1140.737,-37.962,-47.008,179.270,6.157,149.326
C00788=1140.742,-38.212,-46.997,179.267,6.156,149.326
C00789=1140.747,-38.462,-46.985,179.265,6.155,149.327
C00790=1140.752,-38.711,-46.973,179.263,6.155,149.327
C00791=1140.757,-38.961,-46.962,179.260,6.154,149.328
C00792=1140.762,-39.210,-46.951,179.258,6.153,149.329
C00793=1140.768,-39.460,-46.939,179.256,6.153,149.329
C00794=1140.773,-39.710,-46.927,179.253,6.152,149.330
C00795=1140.778,-39.960,-46.916,179.251,6.152,149.330
C00796=1140.784,-40.209,-46.905,179.249,6.151,149.331
C00797=1140.789,-40.459,-46.893,179.246,6.150,149.331
C00798=1140.794,-40.709,-46.882,179.244,6.150,149.332
C00799=1140.799,-40.959,-46.870,179.242,6.149,149.332
C00800=1140.804,-41.208,-46.859,179.239,6.148,149.333
C00801=1140.810,-41.458,-46.847,179.238,6.148,149.334
C00802=1140.815,-41.707,-46.836,179.235,6.148,149.334
C00803=1140.820,-41.958,-46.825,179.233,6.147,149.335
C00804=1140.826,-42.207,-46.814,179.230,6.146,149.335
C00805=1140.831,-42.457,-46.802,179.228,6.146,149.336
C00806=1140.836,-42.706,-46.791,179.226,6.145,149.336
C00807=1140.842,-42.956,-46.779,179.223,6.144,149.337
C00808=1140.847,-43.206,-46.769,179.221,6.144,149.338
C00809=1140.851,-43.455,-46.758,179.219,6.143,149.338
C00810=1140.857,-43.705,-46.746,179.216,6.143,149.339
C00811=1140.862,-43.954,-46.735,179.214,6.142,149.339
C00812=1140.868,-44.204,-46.723,179.212,6.141,149.340
C00813=1140.873,-44.454,-46.712,179.209,6.141,149.340
C00814=1140.878,-44.703,-46.701,179.207,6.140,149.341
C00815=1140.883,-44.953,-46.689,179.204,6.139,149.341
C00816=1140.888,-45.203,-46.678,179.202,6.139,149.342
C00817=1140.894,-45.453,-46.667,179.200,6.139,149.343
C00818=1140.899,-45.702,-46.656,179.198,6.138,149.343
C00819=1140.904,-45.952,-46.645,179.196,6.137,149.343
C00820=1140.909,-46.203,-46.634,179.193,6.137,149.344
C00821=1140.915,-46.452,-46.623,179.191,6.136,149.345
C00822=1140.919,-46.701,-46.611,179.189,6.135,149.345
C00823=1140.925,-46.952,-46.600,179.186,6.135,149.346
C00824=1140.930,-47.201,-46.589,179.184,6.134,149.346
C00825=1140.936,-47.451,-46.577,179.182,6.134,149.347
C00826=1140.942,-47.700,-46.567,179.179,6.133,149.348
C00827=1140.946,-47.950,-46.556,179.177,6.132,149.348
C00828=1140.952,-48.200,-46.544,179.175,6.132,149.348
C00829=1140.957,-48.449,-46.534,179.173,6.132,149.349
C00830=1140.962,-48.699,-46.523,179.170,6.131,149.350
C00831=1140.967,-48.948,-46.511,179.168,6.130,149.350
C00832=1140.973,-49.198,-46.500,179.166,6.130,149.351
C00833=1140.978,-49.448,-46.489,179.163,6.129,149.351
C00834=1140.983,-49.698,-46.479,179.161,6.128,149.352
C00835=1140.989,-49.947,-46.467,179.159,6.128,149.352
C00836=1140.993,-50.197,-46.456,179.156,6.127,149.353
C00837=1141.000,-50.467,-46.444,179.154,6.127,149.353
C00838=1141.005,-50.739,-46.432,179.152,6.126,149.354
C00839=1141.010,-51.010,-46.421,179.149,6.125,149.355
C00840=1141.017,-51.280,-46.409,179.147,6.125,149.355
C00841=1141.021,-51.530,-46.398,179.144,6.124,149.356
C00842=1141.028,-51.779,-46.387,179.142,6.124,149.357
C00843=1141.032,-52.029,-46.375,179.140,6.123,149.357
C00844=1141.037,-52.279,-46.365,179.138,6.123,149.357
C00845=1141.043,-52.528,-46.354,179.135,6.123,149.358
C00846=1141.048,-52.778,-46.343,179.133,6.122,149.359
C00847=1141.054,-53.028,-46.332,179.131,6.121,149.359
C00848=1141.059,-53.278,-46.321,179.128,6.121,149.360
C00849=1141.063,-53.528,-46.310,179.126,6.120,149.360
C00850=1141.069,-53.777,-46.300,179.124,6.119,149.361
C00851=1141.074,-54.027,-46.288,179.121,6.119,149.362
C00852=1141.080,-54.277,-46.278,179.120,6.119,149.362
C00853=1141.085,-54.526,-46.266,179.117,6.118,149.362
C00854=1141.090,-54.776,-46.256,179.115,6.117,149.363
C00855=1141.095,-55.025,-46.245,179.113,6.117,149.364
C00856=1141.101,-55.275,-46.235,179.110,6.116,149.364
C00857=1141.106,-55.525,-46.224,179.108,6.115,149.365
C00858=1141.111,-55.775,-46.212,179.106,6.115,149.365
C00859=1141.117,-56.025,-46.202,179.103,6.114,149.366
C00860=1141.121,-56.274,-46.191,179.102,6.114,149.366
C00861=1141.127,-56.524,-46.180,179.099,6.114,149.367
C00862=1141.132,-56.774,-46.170,179.097,6.113,149.367
C00863=1141.137,-57.023,-46.159,179.095,6.112,149.368
C00864=1141.142,-57.273,-46.148,179.092,6.112,149.369
C00865=1141.148,-57.523,-46.138,179.090,6.111,149.369
C00866=1141.153,-57.773,-46.126,179.088,6.110,149.370
C00867=1141.159,-58.022,-46.116,179.086,6.110,149.370
C00868=1141.163,-58.272,-46.105,179.083,6.110,149.371
C00869=1141.169,-58.521,-46.095,179.081,6.109,149.371
C00870=1141.174,-58.772,-46.084,179.079,6.108,149.372
C00871=1141.179,-59.021,-46.073,179.076,6.108,149.372
C00872=1141.184,-59.271,-46.063,179.074,6.107,149.373
C00873=1141.190,-59.520,-46.052,179.073,6.107,149.373
C00874=1141.195,-59.771,-46.042,179.070,6.107,149.374
C00875=1141.200,-60.019,-46.031,179.068,6.106,149.375
C00876=1141.205,-60.270,-46.020,179.066,6.105,149.375
C00877=1141.211,-60.519,-46.010,179.063,6.105,149.376
C00878=1141.216,-60.769,-45.999,179.061,6.104,149.376
C00879=1141.222,-61.019,-45.988,179.059,6.104,149.377
C00880=1141.227,-61.268,-45.978,179.057,6.103,149.377
C00881=1141.232,-61.519,-45.967,179.054,6.103,149.378
C00882=1141.238,-61.767,-45.956,179.052,6.102,149.378
C00883=1141.243,-62.018,-45.946,179.050,6.102,149.379
C00884=1141.248,-62.267,-45.935,179.047,6.101,149.380
C00885=1141.253,-62.518,-45.925,179.046,6.101,149.380
C00886=1141.259,-62.767,-45.915,179.043,6.100,149.381
C00887=1141.264,-63.017,-45.903,179.041,6.100,149.381
C00888=1141.269,-63.266,-45.893,179.039,6.099,149.382
C00889=1141.275,-63.516,-45.883,179.036,6.098,149.382
C00890=1141.280,-63.766,-45.872,179.034,6.098,149.383
C00891=1141.285,-64.016,-45.862,179.032,6.098,149.383
C00892=1141.290,-64.266,-45.852,179.030,6.097,149.384
C00893=1141.296,-64.515,-45.841,179.028,6.097,149.384
C00894=1141.301,-64.764,-45.830,179.026,6.096,149.385
C00895=1141.306,-65.014,-45.821,179.023,6.095,149.386
C00896=1141.311,-65.264,-45.810,179.021,6.095,149.386
C00897=1141.316,-65.514,-45.800,179.019,6.095,149.387
C00898=1141.322,-65.764,-45.790,179.016,6.094,149.387
C00899=1141.327,-66.013,-45.779,179.014,6.094,149.388
C00900=1141.332,-66.263,-45.768,179.012,6.093,149.388
C00901=1141.338,-66.512,-45.758,179.010,6.093,149.389
C00902=1141.343,-66.762,-45.747,179.008,6.092,149.389
C00903=1141.348,-67.012,-45.737,179.006,6.092,149.390
C00904=1141.354,-67.262,-45.727,179.003,6.091,149.390
C00905=1141.359,-67.512,-45.716,179.001,6.090,149.391
C00906=1141.364,-67.761,-45.706,178.999,6.090,149.392
C00907=1141.370,-68.011,-45.696,178.997,6.090,149.392
C00908=1141.375,-68.261,-45.685,178.995,6.089,149.392
C00909=1141.380,-68.510,-45.676,178.992,6.089,149.393
C00910=1141.385,-68.760,-45.665,178.990,6.088,149.394
C00911=1141.390,-69.010,-45.655,178.988,6.088,149.394
C00912=1141.396,-69.260,-45.645,178.986,6.087,149.395
C00913=1141.402,-69.509,-45.634,178.983,6.087,149.395
C00914=1141.407,-69.760,-45.624,178.981,6.086,149.396
C00915=1141.412,-70.009,-45.614,178.979,6.085,149.396
C00916=1141.418,-70.259,-45.603,178.977,6.086,149.397
C00917=1141.422,-70.509,-45.593,178.975,6.085,149.397
C00918=1141.428,-70.758,-45.583,178.973,6.084,149.398
C00919=1141.433,-71.008,-45.573,178.970,6.083,149.398
C00920=1141.438,-71.258,-45.562,178.968,6.084,149.399
C00921=1141.444,-71.507,-45.552,178.966,6.083,149.400
C00922=1141.450,-71.757,-45.542,178.964,6.082,149.400
C00923=1141.454,-72.007,-45.532,178.962,6.081,149.401
C00924=1141.459,-72.256,-45.522,178.959,6.081,149.401
C00925=1141.465,-72.506,-45.512,178.957,6.081,149.402
C00926=1141.471,-72.755,-45.501,178.955,6.080,149.402
C00927=1141.476,-73.006,-45.491,178.953,6.080,149.403
C00928=1141.481,-73.256,-45.482,178.950,6.079,149.403
C00929=1141.486,-73.505,-45.472,178.949,6.079,149.404
C00930=1141.491,-73.755,-45.461,178.947,6.078,149.404
C00931=1141.497,-74.005,-45.451,178.944,6.078,149.405
C00932=1141.503,-74.254,-45.441,178.942,6.077,149.406
C00933=1141.507,-74.504,-45.431,178.940,6.077,149.406
C00934=1141.512,-74.754,-45.421,178.938,6.076,149.407
C00935=1141.518,-75.003,-45.410,178.935,6.076,149.407
C00936=1141.524,-75.254,-45.401,178.933,6.075,149.408
C00937=1141.529,-75.503,-45.391,178.932,6.075,149.408
C00938=1141.534,-75.753,-45.381,178.929,6.075,149.409
C00939=1141.539,-76.003,-45.371,178.927,6.074,149.409
C00940=1141.545,-76.252,-45.360,178.924,6.073,149.410
C00941=1141.550,-76.524,-45.350,178.922,6.073,149.410
C00942=1141.556,-76.796,-45.339,178.920,6.072,149.411
C00943=1141.562,-77.066,-45.328,178.918,6.072,149.412
C00944=1141.568,-77.338,-45.318,178.915,6.072,149.412
C00945=1141.573,-77.588,-45.308,178.913,6.071,149.413
C00946=1141.579,-77.837,-45.297,178.911,6.070,149.413
C00947=1141.584,-78.088,-45.287,178.909,6.070,149.414
C00948=1141.589,-78.337,-45.278,178.907,6.070,149.414
C00949=1141.595,-78.587,-45.268,178.904,6.069,149.415
C00950=1141.600,-78.837,-45.257,178.902,6.069,149.415
C00951=1141.605,-79.086,-45.248,178.900,6.068,149.416
C00952=1141.610,-79.337,-45.238,178.898,6.068,149.416
C00953=1141.616,-79.586,-45.228,178.896,6.067,149.417
C00954=1141.621,-79.835,-45.218,178.894,6.067,149.418
C00955=1141.626,-80.085,-45.208,178.892,6.067,149.418
C00956=1141.632,-80.335,-45.198,178.890,6.066,149.419
C00957=1141.637,-80.584,-45.189,178.887,6.066,149.419
C00958=1141.642,-80.835,-45.178,178.885,6.065,149.420
C00959=1141.648,-81.085,-45.169,178.883,6.065,149.420
C00960=1141.653,-81.334,-45.159,178.881,6.064,149.421
C00961=1141.659,-81.584,-45.149,178.878,6.064,149.421
C00962=1141.664,-81.833,-45.140,178.876,6.063,149.422
C00963=1141.669,-82.084,-45.129,178.875,6.063,149.422
C00964=1141.674,-82.333,-45.119,178.873,6.062,149.423
C00965=1141.679,-82.583,-45.110,178.870,6.062,149.423
C00966=1141.685,-82.833,-45.100,178.868,6.062,149.424
C00967=1141.690,-83.082,-45.091,178.866,6.061,149.425
C00968=1141.696,-83.332,-45.081,178.864,6.060,149.425
C00969=1141.701,-83.581,-45.071,178.862,6.060,149.426
C00970=1141.706,-83.832,-45.062,178.860,6.060,149.426
C00971=1141.712,-84.082,-45.051,178.857,6.059,149.427
C00972=1141.716,-84.331,-45.042,178.855,6.059,149.427
C00973=1141.722,-84.581,-45.032,178.854,6.059,149.428
C00974=1141.727,-84.830,-45.023,178.851,6.058,149.428
C00975=1141.733,-85.080,-45.013,178.849,6.057,149.429
C00976=1141.739,-85.330,-45.003,178.847,6.057,149.429
C00977=1141.744,-85.580,-44.994,178.845,6.057,149.430
C00978=1141.749,-85.830,-44.983,178.843,6.056,149.430
C00979=1141.754,-86.079,-44.974,178.840,6.056,149.431
C00980=1141.760,-86.329,-44.964,178.839,6.056,149.432
C00981=1141.765,-86.579,-44.955,178.836,6.055,149.432
C00982=1141.770,-86.829,-44.945,178.834,6.054,149.433
C00983=1141.775,-87.078,-44.936,178.833,6.054,149.433
C00984=1141.781,-87.328,-44.926,178.830,6.054,149.434
C00985=1141.786,-87.577,-44.917,178.828,6.053,149.434
C00986=1141.792,-87.828,-44.907,178.826,6.053,149.435
C00987=1141.797,-88.077,-44.897,178.824,6.052,149.435
C00988=1141.802,-88.328,-44.888,178.822,6.052,149.436
C00989=1141.807,-88.577,-44.878,178.819,6.051,149.436
C00990=1141.813,-88.827,-44.868,178.817,6.051,149.437
C00991=1141.818,-89.076,-44.859,178.815,6.050,149.437
C00992=1141.824,-89.326,-44.849,178.813,6.050,149.438
C00993=1141.829,-89.576,-44.840,178.811,6.050,149.438
C00994=1141.834,-89.826,-44.831,178.809,6.049,149.439
C00995=1141.840,-90.076,-44.821,178.807,6.049,149.439
C00996=1141.844,-90.325,-44.812,178.805,6.049,149.440
C00997=1141.850,-90.575,-44.802,178.803,6.048,149.440
C00998=1141.855,-90.824,-44.793,178.801,6.047,149.441
C00999=1141.861,-91.075,-44.783,178.798,6.048,149.442
C01000=1141.866,-91.324,-44.774,178.796,6.047,149.442
C01001=1141.871,-91.574,-44.765,178.794,6.046,149.443
C01002=1141.877,-91.824,-44.755,178.793,6.046,149.443
C01003=1141.882,-92.073,-44.746,178.790,6.045,149.444
C01004=1141.888,-92.323,-44.736,178.788,6.045,149.444
C01005=1141.893,-92.573,-44.727,178.786,6.045,149.445
C01006=1141.899,-92.823,-44.717,178.784,6.044,149.445
C01007=1141.904,-93.072,-44.708,178.782,6.043,149.446
C01008=1141.909,-93.322,-44.699,178.780,6.043,149.446
C01009=1141.915,-93.572,-44.689,178.778,6.043,149.447
C01010=1141.920,-93.822,-44.680,178.775,6.042,149.447
C01011=1141.925,-94.071,-44.671,178.774,6.042,149.448
C01012=1141.930,-94.321,-44.661,178.771,6.042,149.448
C01013=1141.936,-94.571,-44.652,178.769,6.041,149.449
C01014=1141.942,-94.821,-44.643,178.768,6.041,149.449
C01015=1141.946,-95.070,-44.633,178.765,6.040,149.450
C01016=1141.952,-95.320,-44.624,178.763,6.040,149.451
C01017=1141.957,-95.570,-44.615,178.761,6.040,149.451
C01018=1141.963,-95.820,-44.606,178.759,6.039,149.452
C01019=1141.967,-96.069,-44.596,178.757,6.038,149.452
C01020=1141.973,-96.320,-44.586,178.755,6.038,149.452
C01021=1141.979,-96.569,-44.578,178.753,6.038,149.453
C01022=1141.983,-96.819,-44.568,178.750,6.037,149.454
C01023=1141.989,-97.069,-44.558,178.749,6.037,149.454
C01024=1141.994,-97.319,-44.550,178.746,6.036,149.455
C01025=1142.000,-97.568,-44.541,178.745,6.037,149.455
C01026=1142.006,-97.819,-44.531,178.743,6.036,149.456
C01027=1142.010,-98.068,-44.522,178.741,6.035,149.456
C01028=1142.016,-98.318,-44.513,178.738,6.035,149.457
C01029=1142.021,-98.568,-44.503,178.736,6.035,149.457
C01030=1142.027,-98.818,-44.494,178.734,6.034,149.458
C01031=1142.031,-99.067,-44.485,178.732,6.034,149.458
C01032=1142.037,-99.317,-44.476,178.730,6.033,149.459
C01033=1142.043,-99.567,-44.466,178.728,6.032,149.459
C01034=1142.048,-99.817,-44.457,178.726,6.032,149.460
C01035=1142.054,-100.066,-44.449,178.724,6.032,149.460
C01036=1142.059,-100.316,-44.440,178.722,6.032,149.461
C01037=1142.064,-100.565,-44.430,178.720,6.031,149.461
C01038=1142.069,-100.815,-44.421,178.718,6.031,149.462
C01039=1142.075,-101.065,-44.412,178.716,6.031,149.462
C01040=1142.080,-101.315,-44.403,178.714,6.030,149.463
C01041=1142.086,-101.565,-44.394,178.712,6.029,149.463
C01042=1142.091,-101.815,-44.385,178.710,6.030,149.464
C01043=1142.096,-102.065,-44.376,178.708,6.029,149.465
C01044=1142.101,-102.315,-44.367,178.706,6.029,149.465
C01045=1142.107,-102.587,-44.357,178.704,6.028,149.466
C01046=1142.114,-102.859,-44.347,178.701,6.028,149.466
C01047=1142.119,-103.131,-44.337,178.699,6.027,149.467
C01048=1142.125,-103.403,-44.327,178.697,6.026,149.467
C01049=1142.130,-103.653,-44.318,178.695,6.026,149.468
C01050=1142.135,-103.903,-44.309,178.693,6.026,149.468
C01051=1142.140,-104.152,-44.300,178.691,6.026,149.469
C01052=1142.145,-104.402,-44.291,178.689,6.025,149.469
C01053=1142.152,-104.651,-44.282,178.686,6.025,149.470
C01054=1142.157,-104.901,-44.273,178.685,6.025,149.470
C01055=1142.162,-105.151,-44.264,178.683,6.024,149.471
C01056=1142.167,-105.401,-44.255,178.681,6.024,149.471
C01057=1142.173,-105.651,-44.246,178.679,6.023,149.472
C01058=1142.178,-105.901,-44.237,178.677,6.022,149.472
C01059=1142.184,-106.151,-44.228,178.675,6.023,149.473
C01060=1142.189,-106.400,-44.219,178.672,6.022,149.474
C01061=1142.195,-106.650,-44.210,178.671,6.022,149.474
C01062=1142.200,-106.900,-44.201,178.669,6.021,149.475
C01063=1142.205,-107.150,-44.193,178.666,6.021,149.475
C01064=1142.210,-107.399,-44.184,178.665,6.021,149.475
C01065=1142.215,-107.649,-44.175,178.663,6.020,149.476
C01066=1142.221,-107.898,-44.166,178.661,6.020,149.476
C01067=1142.226,-108.148,-44.157,178.658,6.020,149.477
C01068=1142.232,-108.398,-44.148,178.656,6.019,149.478
C01069=1142.237,-108.648,-44.139,178.655,6.019,149.478
C01070=1142.242,-108.898,-44.130,178.652,6.018,149.479
C01071=1142.249,-109.148,-44.122,178.651,6.018,149.479
C01072=1142.254,-109.398,-44.113,178.649,6.017,149.480
C01073=1142.259,-109.648,-44.104,178.646,6.017,149.480
C01074=1142.264,-109.897,-44.096,178.645,6.017,149.481
C01075=1142.269,-110.147,-44.087,178.643,6.016,149.481
C01076=1142.275,-110.396,-44.078,178.641,6.016,149.482
C01077=1142.280,-110.646,-44.069,178.638,6.016,149.482
C01078=1142.285,-110.896,-44.060,178.637,6.016,149.483
C01079=1142.290,-111.146,-44.051,178.634,6.015,149.483
C01080=1142.296,-111.396,-44.042,178.632,6.014,149.484
C01081=1142.302,-111.646,-44.034,178.631,6.014,149.484
C01082=1142.308,-111.896,-44.025,178.628,6.013,149.485
C01083=1142.313,-112.146,-44.016,178.627,6.013,149.485
C01084=1142.318,-112.396,-44.007,178.625,6.013,149.486
C01085=1142.324,-112.645,-43.999,178.623,6.013,149.486
C01086=1142.329,-112.895,-43.990,178.621,6.012,149.487
C01087=1142.334,-113.145,-43.982,178.619,6.011,149.487
C01088=1142.340,-113.395,-43.973,178.617,6.012,149.488
C01089=1142.345,-113.644,-43.964,178.614,6.011,149.488
C01090=1142.350,-113.894,-43.955,178.613,6.011,149.489
C01091=1142.356,-114.144,-43.947,178.611,6.010,149.489
C01092=1142.361,-114.394,-43.938,178.609,6.010,149.490
C01093=1142.367,-114.643,-43.930,178.607,6.010,149.490
C01094=1142.372,-114.893,-43.921,178.605,6.009,149.491
C01095=1142.377,-115.143,-43.912,178.603,6.009,149.491
C01096=1142.382,-115.393,-43.903,178.601,6.008,149.492
C01097=1142.388,-115.643,-43.895,178.599,6.008,149.492
C01098=1142.394,-115.892,-43.886,178.597,6.007,149.493
C01099=1142.399,-116.142,-43.878,178.595,6.007,149.493
C01100=1142.405,-116.391,-43.869,178.593,6.007,149.494
C01101=1142.410,-116.642,-43.861,178.592,6.007,149.494
C01102=1142.414,-116.891,-43.853,178.589,6.006,149.495
C01103=1142.420,-117.141,-43.844,178.587,6.006,149.495
C01104=1142.425,-117.390,-43.835,178.585,6.006,149.496
C01105=1142.431,-117.641,-43.827,178.583,6.005,149.496
C01106=1142.436,-117.891,-43.818,178.581,6.005,149.497
C01107=1142.442,-118.140,-43.809,178.579,6.004,149.497
C01108=1142.447,-118.390,-43.801,178.578,6.004,149.498
C01109=1142.452,-118.640,-43.792,178.575,6.003,149.498
C01110=1142.458,-118.889,-43.784,178.574,6.004,149.499
C01111=1142.464,-119.140,-43.776,178.572,6.003,149.499
C01112=1142.469,-119.390,-43.767,178.570,6.003,149.500
C01113=1142.475,-119.639,-43.758,178.568,6.002,149.500
C01114=1142.479,-119.889,-43.751,178.566,6.001,149.501
C01115=1142.484,-120.139,-43.742,178.564,6.001,149.501
C01116=1142.490,-120.388,-43.733,178.562,6.001,149.502
C01117=1142.496,-120.639,-43.725,178.560,6.001,149.502
C01118=1142.501,-120.888,-43.716,178.558,6.000,149.503
C01119=1142.507,-121.138,-43.708,178.556,6.000,149.503
C01120=1142.512,-121.388,-43.699,178.554,5.999,149.504
C01121=1142.517,-121.638,-43.691,178.553,5.999,149.504
C01122=1142.522,-121.887,-43.683,178.550,5.999,149.505
C01123=1142.528,-122.137,-43.674,178.548,5.999,149.505
C01124=1142.533,-122.387,-43.666,178.546,5.998,149.506
C01125=1142.539,-122.637,-43.658,178.545,5.998,149.506
C01126=1142.544,-122.887,-43.649,178.542,5.998,149.507
C01127=1142.549,-123.136,-43.640,178.541,5.998,149.507
C01128=1142.555,-123.386,-43.633,178.539,5.997,149.508
C01129=1142.560,-123.636,-43.624,178.536,5.996,149.508
C01130=1142.565,-123.886,-43.616,178.535,5.996,149.509
C01131=1142.571,-124.135,-43.607,178.533,5.995,149.509
C01132=1142.577,-124.386,-43.599,178.531,5.995,149.510
C01133=1142.582,-124.635,-43.590,178.529,5.995,149.510
C01134=1142.587,-124.885,-43.583,178.527,5.995,149.511
C01135=1142.592,-125.135,-43.574,178.525,5.994,149.511
C01136=1142.598,-125.385,-43.566,178.523,5.994,149.512
C01137=1142.603,-125.635,-43.557,178.521,5.993,149.512
C01138=1142.609,-125.883,-43.549,178.520,5.993,149.513
C01139=1142.614,-126.134,-43.541,178.517,5.993,149.513
C01140=1142.619,-126.384,-43.532,178.516,5.993,149.514
C01141=1142.625,-126.634,-43.524,178.514,5.992,149.514
C01142=1142.630,-126.883,-43.515,178.512,5.992,149.515
C01143=1142.636,-127.133,-43.508,178.510,5.991,149.515
C01144=1142.641,-127.383,-43.500,178.508,5.991,149.516
C01145=1142.646,-127.633,-43.491,178.506,5.990,149.516
C01146=1142.652,-127.883,-43.483,178.504,5.991,149.517
C01147=1142.657,-128.133,-43.475,178.502,5.990,149.517
C01148=1142.663,-128.382,-43.467,178.501,5.990,149.518
C01149=1142.242,-128.393,-43.510,178.497,5.993,149.519
C01150=1142.237,-128.144,-43.519,178.499,5.994,149.519
C01151=1142.231,-127.893,-43.527,178.501,5.994,149.518
C01152=1142.225,-127.644,-43.535,178.503,5.995,149.518
C01153=1142.221,-127.394,-43.543,178.504,5.994,149.517
C01154=1142.215,-127.145,-43.551,178.507,5.995,149.517
C01155=1142.209,-126.895,-43.560,178.508,5.995,149.516
C01156=1142.204,-126.644,-43.568,178.510,5.996,149.516
C01157=1142.199,-126.395,-43.576,178.512,5.996,149.515
C01158=1142.193,-126.145,-43.584,178.514,5.997,149.515
C01159=1142.188,-125.896,-43.592,178.516,5.997,149.514
C01160=1142.182,-125.645,-43.601,178.518,5.997,149.514
C01161=1142.178,-125.396,-43.609,178.520,5.997,149.514
C01162=1142.172,-125.146,-43.617,178.522,5.998,149.513
C01163=1142.166,-124.896,-43.626,178.523,5.998,149.513
C01164=1142.161,-124.647,-43.634,178.526,5.999,149.512
C01165=1142.155,-124.396,-43.642,178.527,5.999,149.512
C01166=1142.151,-124.147,-43.651,178.529,5.999,149.511
C01167=1142.145,-123.897,-43.658,178.531,5.999,149.511
C01168=1142.140,-123.647,-43.667,178.534,6.000,149.510
C01169=1142.133,-123.397,-43.675,178.536,6.000,149.509
C01170=1142.128,-123.148,-43.684,178.537,6.000,149.509
C01171=1142.123,-122.897,-43.692,178.540,6.001,149.508
C01172=1142.118,-122.648,-43.700,178.541,6.001,149.508
C01173=1142.113,-122.398,-43.709,178.543,6.002,149.507
C01174=1142.107,-122.148,-43.717,178.545,6.002,149.507
C01175=1142.101,-121.899,-43.726,178.547,6.003,149.506
C01176=1142.096,-121.648,-43.734,178.549,6.003,149.506
C01177=1142.091,-121.398,-43.743,178.551,6.003,149.505
C01178=1142.086,-121.150,-43.751,178.553,6.003,149.505
C01179=1142.080,-120.899,-43.759,178.555,6.004,149.504
C01180=1142.075,-120.649,-43.768,178.556,6.004,149.504
C01181=1142.069,-120.400,-43.776,178.559,6.005,149.504
C01182=1142.064,-120.150,-43.785,178.560,6.005,149.503
C01183=1142.059,-119.900,-43.793,178.562,6.005,149.503
C01184=1142.053,-119.651,-43.802,178.564,6.005,149.502
C01185=1142.047,-119.400,-43.810,178.566,6.006,149.502
C01186=1142.042,-119.150,-43.819,178.568,6.007,149.501
C01187=1142.037,-118.902,-43.827,178.570,6.007,149.501
C01188=1142.032,-118.651,-43.835,178.572,6.008,149.500
C01189=1142.027,-118.401,-43.844,178.574,6.007,149.500
C01190=1142.021,-118.152,-43.853,178.576,6.008,149.499
C01191=1142.015,-117.902,-43.861,178.578,6.008,149.499
C01192=1142.010,-117.652,-43.870,178.580,6.009,149.498
C01193=1142.004,-117.403,-43.878,178.581,6.009,149.498
C01194=1141.999,-117.152,-43.886,178.584,6.009,149.497
C01195=1141.994,-116.902,-43.895,178.586,6.009,149.496
C01196=1141.988,-116.653,-43.904,178.588,6.010,149.496
C01197=1141.983,-116.403,-43.913,178.590,6.011,149.495
C01198=1141.977,-116.153,-43.921,178.592,6.011,149.495
C01199=1141.972,-115.903,-43.930,178.594,6.011,149.495
C01200=1141.966,-115.654,-43.938,178.595,6.011,149.494
C01201=1141.961,-115.404,-43.947,178.598,6.012,149.494
C01202=1141.956,-115.153,-43.955,178.599,6.012,149.493
C01203=1141.950,-114.904,-43.964,178.601,6.013,149.493
C01204=1141.945,-114.655,-43.973,178.604,6.014,149.492
C01205=1141.940,-114.405,-43.982,178.605,6.014,149.492
C01206=1141.935,-114.155,-43.991,178.607,6.014,149.491
C01207=1141.928,-113.905,-43.998,178.609,6.014,149.491
C01208=1141.923,-113.655,-44.007,178.611,6.015,149.490
C01209=1141.918,-113.405,-44.016,178.613,6.015,149.489
C01210=1141.913,-113.155,-44.025,178.615,6.015,149.489
C01211=1141.907,-112.906,-44.034,178.617,6.015,149.488
C01212=1141.902,-112.656,-44.042,178.619,6.016,149.488
C01213=1141.897,-112.406,-44.051,178.621,6.017,149.487
C01214=1141.891,-112.156,-44.060,178.623,6.017,149.487
C01215=1141.886,-111.907,-44.068,178.625,6.017,149.486
C01216=1141.880,-111.657,-44.077,178.627,6.017,149.486
C01217=1141.875,-111.407,-44.086,178.629,6.018,149.486
C01218=1141.870,-111.157,-44.095,178.631,6.019,149.485
C01219=1141.865,-110.907,-44.103,178.633,6.019,149.485
C01220=1141.859,-110.658,-44.112,178.635,6.020,149.484
C01221=1141.854,-110.408,-44.121,178.637,6.019,149.483
C01222=1141.849,-110.158,-44.129,178.639,6.020,149.483
C01223=1141.843,-109.908,-44.138,178.641,6.020,149.482
C01224=1141.838,-109.659,-44.147,178.643,6.021,149.482
C01225=1141.832,-109.409,-44.156,178.645,6.021,149.481
C01226=1141.827,-109.159,-44.165,178.647,6.021,149.481
C01227=1141.822,-108.910,-44.174,178.649,6.022,149.480
C01228=1141.816,-108.659,-44.183,178.651,6.022,149.480
C01229=1141.811,-108.410,-44.192,178.653,6.023,149.479
C01230=1141.805,-108.160,-44.200,178.655,6.024,149.479
C01231=1141.800,-107.910,-44.209,178.657,6.023,149.478
C01232=1141.795,-107.660,-44.218,178.659,6.024,149.478
C01233=1141.789,-107.410,-44.226,178.661,6.024,149.477
C01234=1141.784,-107.160,-44.235,178.663,6.025,149.477
C01235=1141.779,-106.911,-44.244,178.665,6.025,149.476
C01236=1141.773,-106.661,-44.253,178.667,6.025,149.476
C01237=1141.767,-106.411,-44.262,178.669,6.026,149.475
C01238=1141.762,-106.161,-44.271,178.671,6.026,149.475
C01239=1141.757,-105.912,-44.280,178.673,6.027,149.474
C01240=1141.752,-105.662,-44.289,178.676,6.027,149.474
C01241=1141.747,-105.412,-44.298,178.677,6.027,149.473
C01242=1141.741,-105.163,-44.306,178.679,6.028,149.473
C01243=1141.736,-104.913,-44.315,178.681,6.028,149.472
C01244=1141.730,-104.663,-44.325,178.683,6.029,149.472
C01245=1141.725,-104.413,-44.334,178.685,6.029,149.471
C01246=1141.720,-104.164,-44.343,178.687,6.029,149.471
C01247=1141.715,-103.914,-44.352,178.689,6.030,149.470
C01248=1141.710,-103.664,-44.361,178.691,6.030,149.470
C01249=1141.704,-103.415,-44.370,178.693,6.030,149.469
C01250=1141.697,-103.142,-44.380,178.696,6.031,149.469
C01251=1141.692,-102.870,-44.390,178.698,6.032,149.468
C01252=1141.686,-102.597,-44.399,178.700,6.031,149.467
C01253=1141.681,-102.325,-44.410,178.702,6.032,149.467
C01254=1141.675,-102.076,-44.419,178.704,6.033,149.466
C01255=1141.670,-101.826,-44.427,178.706,6.033,149.466
C01256=1141.665,-101.576,-44.436,178.708,6.034,149.465
C01257=1141.659,-101.326,-44.446,178.710,6.034,149.465
C01258=1141.653,-101.077,-44.454,178.712,6.034,149.464
C01259=1141.648,-100.827,-44.463,178.715,6.035,149.464
C01260=1141.643,-100.578,-44.473,178.716,6.035,149.463
C01261=1141.637,-100.327,-44.482,178.718,6.035,149.463
C01262=1141.632,-100.078,-44.491,178.721,6.036,149.462
C01263=1141.627,-99.828,-44.500,178.722,6.036,149.462
C01264=1141.622,-99.578,-44.509,178.724,6.037,149.461
C01265=1141.616,-99.328,-44.519,178.727,6.037,149.461
C01266=1141.611,-99.078,-44.528,178.729,6.037,149.460
C01267=1141.606,-98.829,-44.537,178.731,6.038,149.460
C01268=1141.600,-98.578,-44.547,178.732,6.038,149.459
C01269=1141.595,-98.329,-44.556,178.735,6.039,149.459
C01270=1141.589,-98.079,-44.564,178.737,6.039,149.458
C01271=1141.584,-97.830,-44.574,178.739,6.039,149.457
C01272=1141.578,-97.580,-44.583,178.741,6.040,149.457
C01273=1141.573,-97.330,-44.592,178.743,6.041,149.456
C01274=1141.568,-97.080,-44.601,178.745,6.040,149.456
C01275=1141.562,-96.830,-44.610,178.747,6.041,149.456
C01276=1141.557,-96.581,-44.620,178.749,6.042,149.455
C01277=1141.552,-96.331,-44.629,178.751,6.042,149.455
C01278=1141.546,-96.081,-44.638,178.754,6.042,149.454
C01279=1141.541,-95.831,-44.647,178.756,6.043,149.453
C01280=1141.536,-95.582,-44.657,178.757,6.043,149.453
C01281=1141.530,-95.332,-44.666,178.760,6.044,149.452
C01282=1141.525,-95.082,-44.675,178.762,6.045,149.452
C01283=1141.520,-94.833,-44.685,178.763,6.045,149.451
C01284=1141.514,-94.582,-44.694,178.766,6.045,149.451
C01285=1141.509,-94.333,-44.703,178.768,6.046,149.450
C01286=1141.504,-94.083,-44.714,178.770,6.046,149.450
C01287=1141.498,-93.833,-44.722,178.772,6.046,149.449
C01288=1141.493,-93.583,-44.731,178.774,6.047,149.449
C01289=1141.488,-93.334,-44.742,178.776,6.047,149.448
C01290=1141.483,-93.084,-44.750,178.778,6.047,149.448
C01291=1141.477,-92.834,-44.759,178.781,6.048,149.447
C01292=1141.472,-92.585,-44.770,178.782,6.048,149.447
C01293=1141.467,-92.335,-44.778,178.784,6.049,149.446
C01294=1141.461,-92.084,-44.788,178.787,6.050,149.446
C01295=1141.456,-91.835,-44.798,178.789,6.049,149.445
C01296=1141.450,-91.585,-44.807,178.791,6.050,149.444
C01297=1141.445,-91.335,-44.816,178.793,6.051,149.444
C01298=1141.440,-91.086,-44.826,178.795,6.051,149.443
C01299=1141.434,-90.836,-44.835,178.797,6.052,149.443
C01300=1141.429,-90.587,-44.845,178.800,6.052,149.442
C01301=1141.423,-90.336,-44.854,178.801,6.052,149.442
C01302=1141.418,-90.087,-44.864,178.803,6.053,149.441
C01303=1141.412,-89.837,-44.873,178.806,6.053,149.441
C01304=1141.407,-89.587,-44.882,178.807,6.053,149.440
C01305=1141.403,-89.337,-44.892,178.809,6.054,149.440
C01306=1141.397,-89.087,-44.902,178.812,6.054,149.439
C01307=1141.392,-88.838,-44.911,178.814,6.054,149.439
C01308=1141.386,-88.588,-44.921,178.816,6.055,149.438
C01309=1141.381,-88.338,-44.930,178.818,6.056,149.438
C01310=1141.376,-88.088,-44.940,178.820,6.056,149.437
C01311=1141.371,-87.839,-44.949,178.822,6.056,149.436
C01312=1141.365,-87.589,-44.959,178.824,6.057,149.436
C01313=1141.360,-87.340,-44.969,178.826,6.057,149.436
C01314=1141.354,-87.090,-44.978,178.828,6.058,149.435
C01315=1141.349,-86.840,-44.988,178.830,6.059,149.435
C01316=1141.343,-86.590,-44.997,178.833,6.059,149.434
C01317=1141.339,-86.340,-45.007,178.835,6.059,149.433
C01318=1141.333,-86.090,-45.017,178.837,6.060,149.433
C01319=1141.328,-85.841,-45.026,178.839,6.060,149.432
C01320=1141.322,-85.591,-45.036,178.841,6.060,149.432
C01321=1141.317,-85.341,-45.045,178.843,6.061,149.431
C01322=1141.312,-85.092,-45.056,178.846,6.061,149.431
C01323=1141.306,-84.842,-45.065,178.847,6.061,149.430
C01324=1141.301,-84.592,-45.075,178.849,6.062,149.430
C01325=1141.296,-84.342,-45.085,178.852,6.063,149.429
C01326=1141.291,-84.092,-45.094,178.854,6.063,149.429
C01327=1141.285,-83.842,-45.104,178.856,6.063,149.428
C01328=1141.280,-83.593,-45.113,178.858,6.064,149.428
C01329=1141.275,-83.343,-45.123,178.860,6.065,149.427
C01330=1141.269,-83.094,-45.132,178.862,6.064,149.426
C01331=1141.264,-82.844,-45.143,178.864,6.065,149.426
C01332=1141.259,-82.593,-45.152,178.867,6.066,149.425
C01333=1141.254,-82.344,-45.162,178.869,6.067,149.425
C01334=1141.248,-82.094,-45.172,178.870,6.067,149.424
C01335=1141.243,-81.845,-45.181,178.873,6.067,149.424
C01336=1141.237,-81.595,-45.191,178.875,6.068,149.423
C01337=1141.232,-81.345,-45.202,178.877,6.069,149.423
C01338=1141.227,-81.096,-45.210,178.879,6.069,149.422
C01339=1141.222,-80.845,-45.221,178.882,6.069,149.422
C01340=1141.216,-80.596,-45.231,178.884,6.070,149.421
C01341=1141.211,-80.346,-45.240,178.886,6.070,149.421
C01342=1141.205,-80.096,-45.250,178.888,6.070,149.420
C01343=1141.200,-79.847,-45.261,178.890,6.071,149.419
C01344=1141.195,-79.597,-45.271,178.893,6.072,149.419
C01345=1141.189,-79.347,-45.280,178.894,6.071,149.418
C01346=1141.184,-79.097,-45.290,178.896,6.072,149.418
C01347=1141.179,-78.848,-45.300,178.899,6.073,149.417
C01348=1141.173,-78.598,-45.310,178.901,6.073,149.417
C01349=1141.168,-78.348,-45.320,178.903,6.073,149.416
C01350=1141.163,-78.098,-45.330,178.905,6.074,149.416
C01351=1141.158,-77.849,-45.340,178.907,6.075,149.415
C01352=1141.152,-77.599,-45.350,178.910,6.075,149.415
C01353=1141.147,-77.349,-45.359,178.911,6.075,149.414
C01354=1141.141,-77.078,-45.370,178.914,6.076,149.414
C01355=1141.136,-76.807,-45.381,178.916,6.076,149.413
C01356=1141.129,-76.535,-45.392,178.919,6.077,149.412
C01357=1141.124,-76.264,-45.403,178.921,6.077,149.412
C01358=1141.118,-76.014,-45.413,178.923,6.078,149.411
C01359=1141.113,-75.764,-45.424,178.925,6.078,149.411
C01360=1141.108,-75.514,-45.432,178.927,6.079,149.410
C01361=1141.102,-75.265,-45.443,178.930,6.079,149.410
C01362=1141.097,-75.015,-45.453,178.932,6.080,149.409
C01363=1141.092,-74.765,-45.463,178.934,6.080,149.409
C01364=1141.087,-74.516,-45.473,178.936,6.081,149.408
C01365=1141.081,-74.266,-45.483,178.939,6.081,149.407
C01366=1141.075,-74.016,-45.493,178.941,6.082,149.407
C01367=1141.070,-73.766,-45.503,178.942,6.082,149.406
C01368=1141.065,-73.516,-45.514,178.944,6.083,149.406
C01369=1141.060,-73.267,-45.523,178.947,6.083,149.405
C01370=1141.055,-73.017,-45.534,178.949,6.084,149.405
C01371=1141.049,-72.767,-45.544,178.952,6.085,149.404
C01372=1141.044,-72.517,-45.554,178.953,6.085,149.404
C01373=1141.038,-72.268,-45.564,178.956,6.085,149.403
C01374=1141.034,-72.018,-45.574,178.958,6.086,149.403
C01375=1141.028,-71.768,-45.585,178.960,6.087,149.402
C01376=1141.023,-71.519,-45.595,178.962,6.087,149.402
C01377=1141.017,-71.268,-45.605,178.964,6.087,149.401
C01378=1141.012,-71.018,-45.615,178.967,6.088,149.400
C01379=1141.006,-70.769,-45.625,178.969,6.088,149.400
C01380=1141.001,-70.520,-45.635,178.971,6.089,149.400
C01381=1140.996,-70.269,-45.645,178.973,6.089,149.399
C01382=1140.991,-70.020,-45.655,178.975,6.090,149.398
C01383=1140.985,-69.770,-45.666,178.977,6.090,149.398
C01384=1140.980,-69.520,-45.676,178.980,6.091,149.397
C01385=1140.975,-69.271,-45.686,178.982,6.091,149.397
C01386=1140.969,-69.021,-45.697,178.984,6.091,149.396
C01387=1140.965,-68.771,-45.707,178.986,6.092,149.396
C01388=1140.959,-68.522,-45.717,178.989,6.093,149.395
C01389=1140.953,-68.272,-45.727,178.991,6.093,149.395
C01390=1140.948,-68.022,-45.738,178.993,6.093,149.394
C01391=1140.943,-67.772,-45.748,178.995,6.094,149.394
C01392=1140.938,-67.523,-45.759,178.997,6.094,149.393
C01393=1140.933,-67.273,-45.769,179.000,6.095,149.392
C01394=1140.927,-67.024,-45.779,179.002,6.096,149.392
C01395=1140.922,-66.773,-45.790,179.003,6.096,149.391
C01396=1140.916,-66.524,-45.800,179.006,6.096,149.391
C01397=1140.911,-66.274,-45.810,179.008,6.097,149.390
C01398=1140.907,-66.024,-45.820,179.010,6.098,149.390
C01399=1140.901,-65.775,-45.831,179.013,6.098,149.389
C01400=1140.896,-65.524,-45.841,179.015,6.098,149.389
C01401=1140.890,-65.275,-45.851,179.017,6.099,149.388
C01402=1140.885,-65.026,-45.862,179.019,6.100,149.388
C01403=1140.880,-64.776,-45.873,179.022,6.100,149.387
C01404=1140.874,-64.526,-45.883,179.024,6.101,149.386
C01405=1140.869,-64.276,-45.894,179.026,6.102,149.386
C01406=1140.864,-64.026,-45.904,179.028,6.101,149.385
C01407=1140.858,-63.777,-45.914,179.030,6.102,149.385
C01408=1140.853,-63.527,-45.925,179.033,6.103,149.384
C01409=1140.848,-63.278,-45.936,179.035,6.104,149.384
C01410=1140.843,-63.027,-45.946,179.038,6.104,149.383
C01411=1140.837,-62.778,-45.956,179.039,6.104,149.383
C01412=1140.832,-62.528,-45.967,179.041,6.105,149.382
C01413=1140.827,-62.278,-45.977,179.044,6.105,149.381
C01414=1140.821,-62.029,-45.988,179.046,6.106,149.381
C01415=1140.816,-61.779,-45.999,179.048,6.107,149.380
C01416=1140.811,-61.529,-46.009,179.051,6.107,149.380
C01417=1140.806,-61.279,-46.019,179.053,6.107,149.379
C01418=1140.801,-61.030,-46.030,179.055,6.108,149.379
C01419=1140.796,-60.780,-46.041,179.057,6.109,149.378
C01420=1140.790,-60.530,-46.051,179.060,6.109,149.378
C01421=1140.785,-60.280,-46.062,179.062,6.110,149.377
C01422=1140.780,-60.031,-46.073,179.064,6.111,149.377
C01423=1140.774,-59.782,-46.083,179.066,6.110,149.376
C01424=1140.769,-59.532,-46.093,179.068,6.111,149.375
C01425=1140.763,-59.282,-46.105,179.070,6.112,149.375
C01426=1140.758,-59.032,-46.116,179.073,6.112,149.374
C01427=1140.752,-58.783,-46.126,179.075,6.113,149.374
C01428=1140.747,-58.532,-46.136,179.078,6.114,149.373
C01429=1140.742,-58.283,-46.147,179.080,6.114,149.373
C01430=1140.737,-58.033,-46.158,179.082,6.114,149.372
C01431=1140.732,-57.784,-46.168,179.084,6.115,149.372
C01432=1140.727,-57.534,-46.179,179.086,6.115,149.371
C01433=1140.721,-57.284,-46.190,179.089,6.116,149.370
C01434=1140.717,-57.035,-46.201,179.091,6.117,149.370
C01435=1140.711,-56.785,-46.211,179.093,6.117,149.369
C01436=1140.705,-56.535,-46.222,179.095,6.117,149.369
C01437=1140.701,-56.285,-46.234,179.097,6.118,149.368
C01438=1140.695,-56.035,-46.244,179.100,6.119,149.368
C01439=1140.690,-55.785,-46.254,179.102,6.119,149.367
C01440=1140.685,-55.536,-46.265,179.105,6.120,149.367
C01441=1140.680,-55.286,-46.276,179.107,6.120,149.366
C01442=1140.674,-55.037,-46.287,179.109,6.121,149.366
C01443=1140.669,-54.787,-46.298,179.112,6.122,149.365
C01444=1140.663,-54.538,-46.309,179.113,6.122,149.365
C01445=1140.658,-54.287,-46.319,179.115,6.122,149.364
C01446=1140.653,-54.039,-46.330,179.118,6.123,149.363
C01447=1140.648,-53.788,-46.341,179.120,6.124,149.363
C01448=1140.642,-53.538,-46.352,179.122,6.124,149.362
C01449=1140.637,-53.289,-46.363,179.125,6.125,149.362
C01450=1140.632,-53.039,-46.374,179.127,6.126,149.361
C01451=1140.627,-52.790,-46.384,179.129,6.126,149.361
C01452=1140.622,-52.539,-46.395,179.131,6.126,149.360
C01453=1140.616,-52.290,-46.407,179.134,6.127,149.360
C01454=1140.611,-52.040,-46.417,179.136,6.127,149.359
C01455=1140.606,-51.790,-46.428,179.138,6.128,149.359
C01456=1140.600,-51.541,-46.439,179.141,6.129,149.358
C01457=1140.595,-51.291,-46.451,179.143,6.129,149.357
C01458=1140.590,-51.021,-46.462,179.146,6.130,149.357
C01459=1140.584,-50.750,-46.474,179.148,6.131,149.356
C01460=1140.578,-50.479,-46.486,179.150,6.131,149.355
C01461=1140.572,-50.209,-46.498,179.153,6.132,149.355
C01462=1140.567,-49.958,-46.509,179.155,6.132,149.355
C01463=1140.562,-49.709,-46.520,179.158,6.133,149.354
C01464=1140.556,-49.459,-46.531,179.160,6.134,149.353
C01465=1140.551,-49.209,-46.542,179.162,6.134,149.353
C01466=1140.546,-48.960,-46.553,179.165,6.135,149.352
C01467=1140.541,-48.710,-46.564,179.166,6.135,149.352
C01468=1140.536,-48.460,-46.576,179.168,6.136,149.351
C01469=1140.530,-48.211,-46.586,179.171,6.136,149.351
C01470=1140.525,-47.961,-46.597,179.173,6.137,149.350
C01471=1140.520,-47.711,-46.609,179.175,6.138,149.350
C01472=1140.514,-47.461,-46.619,179.178,6.138,149.349
C01473=1140.510,-47.212,-46.630,179.180,6.139,149.348
C01474=1140.504,-46.962,-46.642,179.182,6.139,149.348
C01475=1140.499,-46.712,-46.653,179.185,6.140,149.347
C01476=1140.494,-46.463,-46.664,179.187,6.141,149.347
C01477=1140.489,-46.213,-46.676,179.189,6.141,149.346
C01478=1140.483,-45.963,-46.686,179.192,6.142,149.346
C01479=1140.478,-45.714,-46.697,179.194,6.142,149.345
C01480=1140.473,-45.464,-46.709,179.196,6.143,149.345
C01481=1140.468,-45.215,-46.720,179.199,6.143,149.344
C01482=1140.462,-44.964,-46.731,179.201,6.144,149.343
C01483=1140.457,-44.715,-46.742,179.203,6.145,149.343
C01484=1140.452,-44.466,-46.753,179.206,6.145,149.342
C01485=1140.446,-44.215,-46.765,179.208,6.146,149.342
C01486=1140.441,-43.965,-46.776,179.210,6.146,149.341
C01487=1140.435,-43.716,-46.787,179.213,6.147,149.341
C01488=1140.431,-43.467,-46.799,179.215,6.148,149.340
C01489=1140.426,-43.217,-46.810,179.217,6.148,149.340
C01490=1140.420,-42.966,-46.821,179.220,6.149,149.339
C01491=1140.415,-42.718,-46.832,179.222,6.150,149.338
C01492=1140.409,-42.468,-46.844,179.224,6.150,149.338
C01493=1140.405,-42.218,-46.855,179.226,6.150,149.337
C01494=1140.399,-41.969,-46.867,179.228,6.151,149.337
C01495=1140.394,-41.718,-46.877,179.231,6.152,149.336
C01496=1140.388,-41.469,-46.889,179.233,6.152,149.336
C01497=1140.384,-41.219,-46.901,179.235,6.153,149.335
C01498=1140.378,-40.970,-46.912,179.238,6.154,149.335
C01499=1140.373,-40.720,-46.923,179.240,6.154,149.334
C01500=1140.368,-40.470,-46.935,179.242,6.155,149.333
C01501=1140.363,-40.220,-46.946,179.245,6.155,149.333
C01502=1140.356,-39.971,-46.957,179.247,6.156,149.332
C01503=1140.352,-39.721,-46.969,179.249,6.157,149.332
C01504=1140.346,-39.471,-46.980,179.252,6.157,149.331
C01505=1140.342,-39.221,-46.992,179.254,6.158,149.331
C01506=1140.336,-38.972,-47.003,179.256,6.159,149.330
C01507=1140.331,-38.723,-47.015,179.259,6.159,149.330
C01508=1140.326,-38.473,-47.026,179.261,6.160,149.329
C01509=1140.321,-38.223,-47.038,179.264,6.161,149.329
C01510=1140.315,-37.973,-47.050,179.266,6.161,149.328
C01511=1140.310,-37.724,-47.061,179.268,6.162,149.327
C01512=1140.305,-37.474,-47.072,179.271,6.163,149.327
C01513=1140.300,-37.225,-47.084,179.273,6.163,149.326
C01514=1140.295,-36.975,-47.096,179.275,6.164,149.326
C01515=1140.289,-36.725,-47.107,179.278,6.165,149.325
C01516=1140.284,-36.476,-47.118,179.280,6.165,149.325
C01517=1140.278,-36.226,-47.130,179.282,6.166,149.324
C01518=1140.274,-35.976,-47.142,179.285,6.166,149.324
C01519=1140.268,-35.726,-47.153,179.287,6.166,149.323
C01520=1140.264,-35.477,-47.165,179.289,6.167,149.322
C01521=1140.258,-35.227,-47.176,179.291,6.168,149.322
C01522=1140.252,-34.978,-47.188,179.294,6.168,149.321
C01523=1140.247,-34.728,-47.199,179.296,6.169,149.321
C01524=1140.242,-34.478,-47.211,179.298,6.170,149.320
C01525=1140.237,-34.228,-47.223,179.301,6.170,149.320
C01526=1140.232,-33.978,-47.235,179.303,6.171,149.319
C01527=1140.226,-33.728,-47.246,179.305,6.172,149.319
C01528=1140.221,-33.480,-47.257,179.308,6.172,149.318
C01529=1140.216,-33.230,-47.269,179.310,6.173,149.317
C01530=1140.210,-32.980,-47.281,179.313,6.173,149.317
C01531=1140.206,-32.730,-47.292,179.315,6.174,149.316
C01532=1140.200,-32.481,-47.305,179.317,6.175,149.316
C01533=1140.195,-32.231,-47.317,179.320,6.175,149.315
C01534=1140.190,-31.981,-47.328,179.322,6.176,149.315
C01535=1140.185,-31.731,-47.340,179.324,6.177,149.314
C01536=1140.179,-31.482,-47.352,179.327,6.177,149.313
C01537=1140.174,-31.232,-47.363,179.329,6.178,149.313
C01538=1140.169,-30.982,-47.375,179.331,6.179,149.313
C01539=1140.164,-30.733,-47.387,179.334,6.179,149.312
C01540=1140.158,-30.483,-47.399,179.336,6.180,149.311
C01541=1140.154,-30.234,-47.411,179.338,6.181,149.311
C01542=1140.148,-29.984,-47.422,179.341,6.181,149.310
C01543=1140.143,-29.734,-47.434,179.343,6.182,149.310
C01544=1140.138,-29.485,-47.446,179.346,6.182,149.309
C01545=1140.133,-29.235,-47.458,179.348,6.183,149.309
C01546=1140.127,-28.985,-47.470,179.351,6.185,149.308
C01547=1140.121,-28.736,-47.482,179.353,6.185,149.307
C01548=1140.117,-28.487,-47.494,179.355,6.186,149.307
C01549=1140.112,-28.237,-47.505,179.358,6.187,149.306
C01550=1140.106,-27.987,-47.517,179.360,6.187,149.306
C01551=1140.101,-27.737,-47.529,179.362,6.188,149.305
C01552=1140.096,-27.488,-47.541,179.365,6.189,149.305
C01553=1140.091,-27.238,-47.553,179.367,6.189,149.304
C01554=1140.085,-26.988,-47.565,179.370,6.190,149.304
C01555=1140.080,-26.738,-47.577,179.372,6.190,149.303
C01556=1140.075,-26.489,-47.590,179.374,6.191,149.302
C01557=1140.070,-26.239,-47.601,179.377,6.192,149.302
C01558=1140.065,-25.989,-47.613,179.379,6.192,149.301
C01559=1140.060,-25.740,-47.625,179.381,6.193,149.301
C01560=1140.054,-25.490,-47.637,179.384,6.194,149.300
C01561=1140.049,-25.240,-47.649,179.386,6.194,149.300
C01562=1140.044,-24.970,-47.663,179.388,6.195,149.299
C01563=1140.038,-24.700,-47.675,179.391,6.195,149.298
C01564=1140.033,-24.430,-47.688,179.394,6.197,149.298
C01565=1140.027,-24.160,-47.701,179.397,6.197,149.297
C01566=1140.021,-23.911,-47.713,179.399,6.198,149.297
C01567=1140.016,-23.661,-47.725,179.401,6.199,149.296
C01568=1140.011,-23.411,-47.738,179.404,6.199,149.296
C01569=1140.006,-23.161,-47.750,179.406,6.200,149.295
C01570=1140.001,-22.911,-47.762,179.408,6.201,149.294
C01571=1139.996,-22.662,-47.775,179.411,6.201,149.294
C01572=1139.990,-22.412,-47.787,179.413,6.202,149.293
C01573=1139.985,-22.162,-47.799,179.415,6.203,149.293
C01574=1139.980,-21.913,-47.811,179.418,6.203,149.292
C01575=1139.975,-21.663,-47.822,179.420,6.204,149.292
C01576=1139.970,-21.414,-47.835,179.423,6.205,149.291
C01577=1139.964,-21.164,-47.847,179.425,6.206,149.291
C01578=1139.959,-20.915,-47.859,179.428,6.207,149.290
C01579=1139.954,-20.665,-47.871,179.430,6.207,149.290
C01580=1139.949,-20.415,-47.884,179.433,6.208,149.289
C01581=1139.943,-20.165,-47.896,179.435,6.209,149.288
C01582=1139.938,-19.916,-47.908,179.437,6.209,149.288
C01583=1139.933,-19.666,-47.920,179.440,6.210,149.287
C01584=1139.928,-19.417,-47.933,179.442,6.211,149.287
C01585=1139.922,-19.167,-47.945,179.444,6.211,149.286
C01586=1139.917,-18.918,-47.957,179.447,6.212,149.286
C01587=1139.912,-18.668,-47.970,179.449,6.213,149.285
C01588=1139.907,-18.418,-47.982,179.452,6.213,149.284
C01589=1139.902,-18.168,-47.995,179.454,6.215,149.284
C01590=1139.897,-17.918,-48.007,179.457,6.215,149.283
C01591=1139.891,-17.669,-48.019,179.459,6.216,149.283
C01592=1139.886,-17.420,-48.032,179.461,6.217,149.282
C01593=1139.881,-17.170,-48.044,179.464,6.217,149.282
C01594=1139.876,-16.920,-48.056,179.466,6.218,149.281
C01595=1139.870,-16.671,-48.068,179.468,6.219,149.281
C01596=1139.865,-16.421,-48.081,179.471,6.219,149.280
C01597=1139.861,-16.171,-48.094,179.473,6.220,149.279
C01598=1139.855,-15.921,-48.106,179.476,6.221,149.279
C01599=1139.850,-15.672,-48.118,179.479,6.222,149.278
C01600=1139.845,-15.423,-48.131,179.481,6.223,149.278
C01601=1139.840,-15.173,-48.143,179.483,6.223,149.277
C01602=1139.834,-14.923,-48.155,179.486,6.224,149.277
C01603=1139.829,-14.674,-48.168,179.488,6.225,149.276
C01604=1139.824,-14.423,-48.180,179.491,6.225,149.276
C01605=1139.819,-14.174,-48.193,179.493,6.226,149.275
C01606=1139.814,-13.924,-48.206,179.495,6.227,149.275
C01607=1139.808,-13.675,-48.219,179.498,6.227,149.274
C01608=1139.803,-13.425,-48.231,179.500,6.229,149.273
C01609=1139.798,-13.176,-48.243,179.503,6.229,149.273
C01610=1139.793,-12.926,-48.256,179.505,6.230,149.272
C01611=1139.788,-12.677,-48.269,179.507,6.231,149.272
C01612=1139.783,-12.427,-48.281,179.510,6.231,149.271
C01613=1139.778,-12.177,-48.293,179.512,6.232,149.271
C01614=1139.772,-11.928,-48.306,179.514,6.233,149.270
C01615=1139.767,-11.678,-48.319,179.517,6.233,149.269
C01616=1139.762,-11.428,-48.332,179.520,6.235,149.269
C01617=1139.757,-11.178,-48.344,179.522,6.235,149.269
C01618=1139.752,-10.929,-48.357,179.525,6.236,149.268
C01619=1139.746,-10.680,-48.369,179.527,6.237,149.267
C01620=1139.742,-10.430,-48.382,179.530,6.237,149.267
C01621=1139.736,-10.180,-48.395,179.532,6.238,149.266
C01622=1139.731,-9.931,-48.408,179.534,6.239,149.266
C01623=1139.726,-9.682,-48.420,179.537,6.239,149.265
C01624=1139.721,-9.431,-48.433,179.539,6.241,149.265
C01625=1139.716,-9.182,-48.445,179.542,6.242,149.264
C01626=1139.710,-8.932,-48.459,179.544,6.242,149.263
C01627=1139.705,-8.683,-48.471,179.546,6.243,149.263
C01628=1139.700,-8.433,-48.484,179.549,6.243,149.262
C01629=1139.695,-8.183,-48.497,179.551,6.244,149.262
C01630=1139.690,-7.934,-48.509,179.554,6.246,149.261
C01631=1139.684,-7.684,-48.522,179.557,6.246,149.261
C01632=1139.680,-7.434,-48.535,179.559,6.247,149.260
C01633=1139.675,-7.185,-48.548,179.561,6.248,149.260
C01634=1139.669,-6.936,-48.561,179.564,6.248,149.259
C01635=1139.664,-6.686,-48.574,179.566,6.249,149.259
C01636=1139.659,-6.436,-48.587,179.569,6.249,149.258
C01637=1139.654,-6.187,-48.599,179.571,6.251,149.257
C01638=1139.648,-5.937,-48.613,179.573,6.252,149.257
C01639=1139.644,-5.687,-48.626,179.576,6.252,149.256
C01640=1139.638,-5.438,-48.638,179.578,6.253,149.256
C01641=1139.633,-5.188,-48.651,179.581,6.253,149.255
C01642=1139.627,-4.939,-48.664,179.583,6.254,149.255
C01643=1139.623,-4.689,-48.677,179.586,6.256,149.254
C01644=1139.618,-4.439,-48.690,179.589,6.256,149.253
C01645=1139.612,-4.190,-48.703,179.591,6.257,149.253
C01646=1139.607,-3.940,-48.716,179.593,6.258,149.253
C01647=1139.602,-3.690,-48.728,179.596,6.258,149.252
C01648=1139.596,-3.441,-48.742,179.598,6.260,149.251
C01649=1139.592,-3.191,-48.754,179.601,6.260,149.251
C01650=1139.587,-2.942,-48.767,179.603,6.261,149.250
C01651=1139.581,-2.692,-48.780,179.605,6.262,149.250
C01652=1139.576,-2.442,-48.793,179.608,6.262,149.249
C01653=1139.571,-2.192,-48.806,179.610,6.263,149.249
C01654=1139.566,-1.944,-48.820,179.613,6.265,149.248
C01655=1139.561,-1.694,-48.833,179.616,6.265,149.247
C01656=1139.555,-1.444,-48.846,179.618,6.266,149.247
C01657=1139.551,-1.194,-48.859,179.620,6.266,149.246
C01658=1139.545,-0.944,-48.872,179.623,6.267,149.246
C01659=1139.540,-0.695,-48.885,179.625,6.269,149.245
C01660=1139.536,-0.446,-48.898,179.628,6.269,149.245
C01661=1139.530,-0.196,-48.912,179.630,6.270,149.244
C01662=1139.525,0.053,-48.924,179.633,6.270,149.243
C01663=1139.519,0.304,-48.938,179.635,6.271,149.243
C01664=1139.514,0.553,-48.950,179.638,6.273,149.243
C01665=1139.509,0.803,-48.965,179.641,6.273,149.242
C01666=1139.504,1.072,-48.978,179.643,6.274,149.241
C01667=1139.498,1.342,-48.992,179.646,6.275,149.241
C01668=1139.493,1.611,-49.007,179.648,6.276,149.240
C01669=1139.487,1.880,-49.020,179.651,6.276,149.240
C01670=1139.482,2.131,-49.034,179.654,6.278,149.239
C01671=1139.477,2.379,-49.047,179.656,6.278,149.238
C01672=1139.472,2.630,-49.061,179.658,6.279,149.238
C01673=1139.466,2.879,-49.074,179.661,6.280,149.237
C01674=1139.462,3.129,-49.088,179.664,6.281,149.237
C01675=1139.456,3.378,-49.100,179.666,6.282,149.236
C01676=1139.451,3.628,-49.114,179.669,6.282,149.236
C01677=1139.446,3.877,-49.127,179.671,6.283,149.235
C01678=1139.440,4.127,-49.140,179.673,6.284,149.235
C01679=1139.436,4.377,-49.153,179.676,6.285,149.234
C01680=1139.430,4.626,-49.167,179.678,6.286,149.234
C01681=1139.426,4.876,-49.180,179.681,6.287,149.233
C01682=1139.420,5.125,-49.194,179.683,6.287,149.232
C01683=1139.416,5.375,-49.207,179.686,6.289,149.232
C01684=1139.410,5.624,-49.220,179.689,6.289,149.231
C01685=1139.405,5.874,-49.235,179.691,6.290,149.231
C01686=1139.400,6.123,-49.247,179.693,6.291,149.230
C01687=1139.395,6.374,-49.261,179.696,6.292,149.230
C01688=1139.390,6.622,-49.274,179.699,6.293,149.229
C01689=1139.384,6.873,-49.288,179.701,6.293,149.229
C01690=1139.379,7.122,-49.302,179.703,6.294,149.228
C01691=1139.374,7.372,-49.315,179.706,6.296,149.228
C01692=1139.369,7.621,-49.329,179.709,6.296,149.227
C01693=1139.364,7.871,-49.341,179.711,6.297,149.226
C01694=1139.359,8.120,-49.355,179.713,6.298,149.226
C01695=1139.354,8.370,-49.369,179.716,6.299,149.225
C01696=1139.349,8.619,-49.382,179.719,6.300,149.225
C01697=1139.343,8.869,-49.396,179.721,6.300,149.224
C01698=1139.338,9.118,-49.410,179.723,6.301,149.224
C01699=1139.333,9.368,-49.423,179.726,6.303,149.223
C01700=1139.328,9.618,-49.437,179.729,6.303,149.223
C01701=1139.323,9.868,-49.450,179.731,6.304,149.222
C01702=1139.318,10.117,-49.464,179.734,6.305,149.221
C01703=1139.312,10.367,-49.477,179.736,6.306,149.221
C01704=1139.308,10.616,-49.491,179.739,6.307,149.220
C01705=1139.302,10.866,-49.504,179.741,6.307,149.220
C01706=1139.297,11.115,-49.518,179.744,6.309,149.219
C01707=1139.292,11.364,-49.532,179.746,6.310,149.219
C01708=1139.287,11.614,-49.545,179.749,6.310,149.218
C01709=1139.282,11.864,-49.559,179.751,6.311,149.218
C01710=1139.277,12.114,-49.573,179.754,6.312,149.217
C01711=1139.272,12.363,-49.587,179.756,6.313,149.217
C01712=1139.267,12.612,-49.600,179.759,6.314,149.216
C01713=1139.262,12.862,-49.614,179.762,6.315,149.215
C01714=1139.257,13.112,-49.628,179.764,6.316,149.215
C01715=1139.251,13.361,-49.642,179.766,6.317,149.214
C01716=1139.246,13.611,-49.655,179.769,6.318,149.214
C01717=1139.241,13.860,-49.669,179.772,6.319,149.213
C01718=1139.236,14.110,-49.683,179.774,6.319,149.213
C01719=1139.231,14.360,-49.697,179.776,6.320,149.212
C01720=1139.225,14.609,-49.711,179.779,6.322,149.212
C01721=1139.221,14.859,-49.724,179.782,6.322,149.211
C01722=1139.216,15.108,-49.738,179.784,6.323,149.211
C01723=1139.210,15.358,-49.752,179.787,6.325,149.210
C01724=1139.205,15.608,-49.766,179.789,6.325,149.209
C01725=1139.200,15.857,-49.780,179.792,6.326,149.209
C01726=1139.195,16.106,-49.794,179.795,6.327,149.208
C01727=1139.190,16.356,-49.807,179.797,6.328,149.208
C01728=1139.185,16.606,-49.821,179.799,6.329,149.207
C01729=1139.180,16.855,-49.835,179.802,6.330,149.207
C01730=1139.175,17.105,-49.850,179.805,6.331,149.206
C01731=1139.170,17.355,-49.864,179.807,6.332,149.206
C01732=1139.164,17.604,-49.877,179.809,6.332,149.205
C01733=1139.160,17.854,-49.891,179.812,6.334,149.205
C01734=1139.155,18.103,-49.905,179.815,6.334,149.204
C01735=1139.149,18.352,-49.919,179.817,6.335,149.204
C01736=1139.144,18.602,-49.933,179.820,6.336,149.203
C01737=1139.139,18.852,-49.947,179.822,6.337,149.202
C01738=1139.133,19.101,-49.961,179.825,6.338,149.202
C01739=1139.128,19.351,-49.975,179.827,6.339,149.201
C01740=1139.123,19.601,-49.989,179.830,6.340,149.201
C01741=1139.118,19.850,-50.004,179.832,6.341,149.200
C01742=1139.113,20.099,-50.017,179.835,6.342,149.200
C01743=1139.109,20.349,-50.031,179.838,6.343,149.199
C01744=1139.104,20.599,-50.045,179.840,6.343,149.199
C01745=1139.099,20.848,-50.060,179.843,6.345,149.198
C01746=1139.093,21.097,-50.074,179.845,6.345,149.198
C01747=1139.088,21.347,-50.088,179.848,6.347,149.197
C01748=1139.083,21.597,-50.102,179.851,6.348,149.196
C01749=1139.078,21.846,-50.116,179.853,6.348,149.196
C01750=1139.073,22.095,-50.130,179.856,6.350,149.196
C01751=1139.068,22.345,-50.145,179.858,6.350,149.195
C01752=1139.063,22.595,-50.159,179.860,6.351,149.194
C01753=1139.058,22.845,-50.173,179.864,6.352,149.194
C01754=1139.052,23.094,-50.187,179.866,6.353,149.193
C01755=1139.047,23.343,-50.201,179.868,6.354,149.193
C01756=1139.042,23.593,-50.216,179.871,6.355,149.192
C01757=1139.038,23.843,-50.230,179.873,6.356,149.192
C01758=1139.033,24.092,-50.244,179.876,6.357,149.191
C01759=1139.027,24.341,-50.258,179.879,6.358,149.191
C01760=1139.022,24.591,-50.272,179.881,6.359,149.190
C01761=1139.017,24.841,-50.287,179.884,6.360,149.189
C01762=1139.012,25.091,-50.301,179.886,6.361,149.189
C01763=1139.007,25.340,-50.315,179.889,6.362,149.188
C01764=1139.001,25.590,-50.330,179.892,6.363,149.188
C01765=1138.996,25.839,-50.344,179.894,6.364,149.187
C01766=1138.991,26.088,-50.359,179.896,6.365,149.187
C01767=1138.986,26.338,-50.373,179.899,6.366,149.186
C01768=1138.981,26.588,-50.388,179.902,6.367,149.186
C01769=1138.976,26.838,-50.402,179.904,6.369,149.185
C01770=1138.971,27.106,-50.417,179.907,6.369,149.185
C01771=1138.965,27.375,-50.432,179.910,6.370,149.184
C01772=1138.959,27.644,-50.448,179.912,6.371,149.183
C01773=1138.954,27.913,-50.464,179.916,6.372,149.183
C01774=1138.949,28.163,-50.478,179.918,6.373,149.182
C01775=1138.944,28.412,-50.493,179.921,6.375,149.182
C01776=1138.939,28.662,-50.507,179.923,6.375,149.181
C01777=1138.933,28.911,-50.522,179.925,6.376,149.181
C01778=1138.928,29.160,-50.536,179.928,6.378,149.180
C01779=1138.924,29.410,-50.551,179.931,6.378,149.180
C01780=1138.919,29.660,-50.565,179.934,6.380,149.179
C01781=1138.914,29.909,-50.580,179.936,6.381,149.179
C01782=1138.909,30.159,-50.594,179.939,6.382,149.178
C01783=1138.903,30.409,-50.609,179.941,6.383,149.178
C01784=1138.898,30.658,-50.623,179.944,6.383,149.177
C01785=1138.894,30.907,-50.638,179.947,6.385,149.176
C01786=1138.889,31.157,-50.653,179.949,6.385,149.176
C01787=1138.883,31.406,-50.667,179.952,6.387,149.175
C01788=1138.878,31.656,-50.682,179.954,6.388,149.175
C01789=1138.873,31.905,-50.696,179.956,6.388,149.174
C01790=1138.868,32.155,-50.711,179.960,6.390,149.174
C01791=1138.863,32.404,-50.726,179.962,6.390,149.173
C01792=1138.858,32.654,-50.741,179.965,6.392,149.173
C01793=1138.853,32.903,-50.756,179.967,6.393,149.172
C01794=1138.848,33.153,-50.770,179.970,6.394,149.172
C01795=1138.843,33.403,-50.784,179.972,6.395,149.171
C01796=1138.838,33.652,-50.800,179.975,6.395,149.171
C01797=1138.833,33.902,-50.814,179.978,6.397,149.170
C01798=1138.828,34.151,-50.829,179.980,6.398,149.169
C01799=1138.822,34.401,-50.844,179.983,6.399,149.169
C01800=1138.817,34.651,-50.858,179.985,6.400,149.169
C01801=1138.813,34.900,-50.873,179.988,6.401,149.168
C01802=1138.807,35.150,-50.888,179.990,6.402,149.167
C01803=1138.802,35.399,-50.903,179.993,6.403,149.167
C01804=1138.797,35.649,-50.917,179.996,6.404,149.166
C01805=1138.792,35.898,-50.933,179.998,6.405,149.166
C01806=1138.787,36.148,-50.947,-179.999,6.407,149.165
C01807=1138.782,36.397,-50.962,-179.997,6.407,149.165
C01808=1138.777,36.647,-50.977,-179.994,6.409,149.164
C01809=1138.772,36.896,-50.992,-179.992,6.409,149.164
C01810=1138.767,37.146,-51.006,-179.988,6.411,149.163
C01811=1138.762,37.395,-51.022,-179.986,6.412,149.163
C01812=1138.757,37.644,-51.037,-179.983,6.413,149.162
C01813=1138.751,37.894,-51.052,-179.981,6.414,149.162
C01814=1138.747,38.143,-51.067,-179.979,6.414,149.161
C01815=1138.742,38.393,-51.081,-179.976,6.416,149.161
C01816=1138.736,38.642,-51.097,-179.973,6.417,149.160
C01817=1138.731,38.892,-51.111,-179.970,6.418,149.160
C01818=1138.726,39.141,-51.126,-179.968,6.419,149.159
C01819=1138.721,39.390,-51.141,-179.965,6.420,149.158
C01820=1138.716,39.640,-51.156,-179.963,6.421,149.158
C01821=1138.711,39.890,-51.171,-179.960,6.423,149.158
C01822=1138.706,40.139,-51.186,-179.957,6.423,149.157
C01823=1138.701,40.389,-51.201,-179.955,6.425,149.156
C01824=1138.696,40.638,-51.216,-179.952,6.425,149.156
C01825=1138.691,40.888,-51.232,-179.949,6.427,149.155
C01826=1138.686,41.138,-51.246,-179.947,6.428,149.155
C01827=1138.681,41.387,-51.262,-179.944,6.429,149.154
C01828=1138.676,41.636,-51.277,-179.942,6.430,149.154
C01829=1138.671,41.886,-51.292,-179.939,6.431,149.153
C01830=1138.666,42.135,-51.307,-179.936,6.432,149.153
C01831=1138.661,42.385,-51.322,-179.934,6.434,149.152
C01832=1138.656,42.634,-51.337,-179.931,6.434,149.152
C01833=1138.650,42.884,-51.352,-179.928,6.436,149.151
C01834=1138.646,43.134,-51.368,-179.926,6.436,149.151
C01835=1138.641,43.383,-51.383,-179.923,6.438,149.150
C01836=1138.636,43.632,-51.398,-179.921,6.439,149.149
C01837=1138.631,43.881,-51.414,-179.918,6.440,149.149
C01838=1138.625,44.131,-51.429,-179.916,6.441,149.149
C01839=1138.620,44.381,-51.444,-179.912,6.442,149.148
C01840=1138.615,44.630,-51.459,-179.910,6.443,149.147
C01841=1138.611,44.880,-51.475,-179.908,6.445,149.147
C01842=1138.606,45.129,-51.490,-179.905,6.445,149.146
